// TIA Portal project "V6_V2.0" (V16)

(* hardware
DEVICE "S7-1200 station_1"  S7-1200 Station
   slot 0: "Rack_0"  S7-1200 Rack  Rack  V1.0
   slot 1: "PLC_Slave"  CPU 1214C DC/DC/DC  6ES7 214-1AG40-0XB0  V4.4
   slot 2: "DI 8/DQ 8x24VDC_1"  6ES7 223-1BH32-0XB0  V2.0
   slot 101: "CM 1241 (RS422/485)_1"  6ES7 241-1CH32-0XB0  V2.2
   slot 102: "CM 1241 (RS422/485)_2"  6ES7 241-1CH32-0XB0  V2.2
   slot 103: "CM 1241 (RS422/485)_3"  6ES7 241-1CH32-0XB0  V2.2
DEVICE "ADMIN_CONTROL_SYSTEM"  KTP700 Basic PN
   slot 0: "HMI_1"  KTP700 Basic PN  6AV2 123-2GB03-0AX0  15.1.0.0
   slot 1: "HMI_RT_1"  KTP700 Basic PN  6AV2 123-2GB03-0AX0  15.1.0.0
   slot 5: "HMI_1.IE_CP_1"  PROFINET Interface  15.0.1.0
      slot 1: "PROFINET Interface_1"  PROFINET Interface
         slot 1: "Port_1"  Port
DEVICE "PC_SEVER"  SIMATIC PC station
   slot 0: "SIMATIC PC station"  Rail  SIMATIC PC-Station  V1.0
      slot 125: "Stationmanager"  Station_Manager  V6.0.4
   slot 1: "HMI_RT_2"  WinCC RT Professional  6AV2 105-0xxxx-xxxx  16.0.0.0
   slot 2: "IE general_1"  IE General  IE_CP  V8.2.0
*)

// ===== PLC "PLC_Slave"  CPU 1214C DC/DC/DC =====

VAR_GLOBAL   // PLC tag table "Default tag table"
   "Sensor_Coun" AT %M100.0 : Bool;
   "Sensor_coun_Check" AT %M100.1 : Bool;
   "Tag_1" AT %I20.1 : Bool;
END_VAR

VAR_GLOBAL   // PLC tag table "SS"
   "SS01" AT %I0.1 : Bool;   // ht tren
   "SS02" AT %I0.2 : Bool;
   "SS03" AT %I0.3 : Bool;   // thang_ngan
   "SS04" AT %I0.4 : Bool;   // thang_dai
   "SS05" AT %I0.5 : Bool;
   "SS06" AT %I0.6 : Bool;
   "SS07" AT %I0.7 : Bool;   // mam_Chot_duoi
   "SS08" AT %I1.0 : Bool;   // mam_chot_tren
   "SS09" AT %I1.1 : Bool;
   "SS10" AT %I1.2 : Bool;
   "SS11" AT %I1.3 : Bool;
   "SS12" AT %I1.4 : Bool;   // xoay_trong
   "SS13" AT %I1.5 : Bool;   // xoay_ngoai
   "SS14" AT %I1.6 : Bool;
   "SS15" AT %I1.7 : Bool;
   "NANG" AT %Q0.1 : Bool;
   "XOAY" AT %Q0.0 : Bool;
   "SS00" AT %I0.0 : Bool;   // ht duoi
   "SS16" AT %I2.0 : Bool;
   "SS17" AT %I2.1 : Bool;
   "SS18" AT %I2.2 : Bool;
   "SS19" AT %I2.3 : Bool;
   "SS20" AT %I2.4 : Bool;
END_VAR

DATA_BLOCK "ControlSystems_DB"   // DB10
{ S7_Optimized_Access := 'FALSE' }
VERSION : 0.1
// stored: InstanceOfName ControlSystems
"ControlSystems"
BEGIN
END_DATA_BLOCK

DATA_BLOCK "MANUAL_DB"   // DB11
{ S7_Optimized_Access := 'TRUE' }
VERSION : 0.1
// stored: InstanceOfName MANUAL
"MANUAL"
BEGIN
END_DATA_BLOCK

DATA_BLOCK "AUTO_DB"   // DB12
{ S7_Optimized_Access := 'TRUE' }
VERSION : 0.1
// stored: InstanceOfName AUTO
"AUTO"
BEGIN
END_DATA_BLOCK

DATA_BLOCK "AutoMode1_DB"   // DB20
{ S7_Optimized_Access := 'TRUE' }
VERSION : 0.1
// stored: InstanceOfName AutoMode1
"AutoMode1"
BEGIN
END_DATA_BLOCK

DATA_BLOCK "AutoMode2_DB"   // DB21
{ S7_Optimized_Access := 'TRUE' }
VERSION : 0.1
// stored: InstanceOfName AutoMode2
"AutoMode2"
BEGIN
END_DATA_BLOCK

DATA_BLOCK "DataSetUp"   // DB24
{ S7_Optimized_Access := 'FALSE' }
VERSION : 0.1
   VAR
      SPEED : Struct
         ELEVATOR : Struct
            Speed_RunManual : Int := 500;
            Speed_StartUp : Int := 500;
            Speed_R1 : Int;
            Speed_R2 : Int;
            Speed_Stop : Int;
         END_STRUCT;
         Cart_Pallet : Struct
            Speed_RunManual : Int := 500;
            Speed_StartUp : Int := 500;
            Speed_R1 : Int;
            Speed_R2 : Int;
            Speed_Stop : Int;
         END_STRUCT;
      END_STRUCT;
      MODE : Struct
         Manual_Auto : Bool;
         ModeNumber : Int;
         AUTO : Struct
            "Auto/Mode1_Mode2" : Bool;
            MODE2 : Struct
               "Mode2/Mode1_Mode2" : Bool;
            END_STRUCT;
         END_STRUCT;
      END_STRUCT;
      DATA__STATUS_MODBUSRTU : Struct
         ELAVATOR : Struct
            StatusUp : Word := 16#0004;
            StartusDown : Word := 16#0002;
         END_STRUCT;
         CART : Struct
            StatusUp : Word := 16#0004;
            StartusDown : Word := 16#0002;
         END_STRUCT;
      END_STRUCT;
   END_VAR
BEGIN
END_DATA_BLOCK

DATA_BLOCK "ControlAtElevator_DB"   // DB25
{ S7_Optimized_Access := 'FALSE' }
VERSION : 0.1
// stored: InstanceOfName ControlAtElevator
"ControlAtElevator"
BEGIN
END_DATA_BLOCK

DATA_BLOCK "Data_ADMIN_HMI"   // DB26
{ S7_Optimized_Access := 'FALSE' }
VERSION : 0.1
   VAR
      OKE : Bool;
      blink_Manual : Bool;
      blink_Auto : Bool;
      blink_Cancel : Bool;
      blink_Setup : Bool;
      blink_Back : Bool;
      blink_Position : Bool;
      Position : Struct
         "201" : Bool;
         "202" : Bool;
         "101" : Bool;
         "102" : Bool;
      END_STRUCT;
      CheckPosition : Struct
         "201" : Bool;
         "202" : Bool;
         "101" : Bool;
         "102" : Bool;
      END_STRUCT;
      PositionNumber : Int;
   END_VAR
BEGIN
END_DATA_BLOCK

DATA_BLOCK "POSITION_DB"   // DB27
{ S7_Optimized_Access := 'TRUE' }
VERSION : 0.1
// stored: InstanceOfName POSITION
"POSITION"
BEGIN
END_DATA_BLOCK

DATA_BLOCK "ModbusRtu_DB"   // DB63
{ S7_Optimized_Access := 'TRUE' }
VERSION : 0.1
// stored: InstanceOfName ModbusRtu
"ModbusRtu"
BEGIN
END_DATA_BLOCK

DATA_BLOCK "FunctionsControlSystems_DB"   // DB65
{ S7_Optimized_Access := 'TRUE' }
VERSION : 0.1
// stored: InstanceOfName FunctionsControlSystems
"FunctionsControlSystems"
BEGIN
END_DATA_BLOCK

// folder: Control

DATA_BLOCK "Data_Control"   // DB5
{ S7_Optimized_Access := 'FALSE' }
VERSION : 0.1
   VAR
      AUTO : Struct
         "Auto.Mode1" : Struct
            STEP_E : Int;
            STEP_HP : Int;
            STEP_TR : Int;
         END_STRUCT;
         "Auto.Mode2_Mode1" : Struct
            Step_ParkingCar : Int;
            Step_GetCar : Int;
         END_STRUCT;
      END_STRUCT;
      Stop : Bool;
      START : Bool;
      RST : Bool;
      Auto_Manual : Bool;
      "Auto.Mode1_Mode2" : Bool;
      "Auto.Mode2_Mode1" : Bool;
      ERROR : Bool;
      ERRORNumber : Int;
      ModeAction : Int;
      ModeNumber : Int;
      SlotIDFrom : Int;
      SlotIDTO : Int;
      Lock : Bool;
      "Auto.ACTION" : Struct
         Elevator : Bool;
         Elevator_2 : Bool;
         HookPallet : Bool;
         HookPallet_2 : Bool;
         TableRotation : Bool;
         TableRotation_2 : Bool;
      END_STRUCT;
      Elevator : Struct
         Start : Bool;
         Done : Bool;
         Running : Bool;
         Error : Bool;
         UP : Bool;
         DOWN : Bool;
         SpeedManual : Int := 500;
         SpeedStartup : Int := 700;   // 7
         Speed1_Auto : Int := 2500;   // 25
         Speed2_Auto : Int := 1000;   // 10
         SpeedStop : Int := 500;   // 5
         "Step" : Int;
         DataSPEEDLift_INVT : Int;
         DataSTATUSControl_INVT : Word;
         DataStatusUPControl_Setup : Word := 16#0004;
         DataStatusDOWNControl_Setup : Word := 16#0002;
         FloorAddressControlNumber : Int := 1;
         FloorAddressControlNumber_Check : Int;
         FloorAddressReal : Int := 1;
         FloorAddressReal_Check : Int := 1;
         FloorAddressReal_Sub_FloorAddressControlNumber : Int;
         time_Run_one : Time := T#2s;   // 2s
         time_Run_Two : Time := T#8s;   // 8s
         time_Run_Three : Time;
      END_STRUCT;
      HookPallet : Struct
         Start : Bool;
         Done : Bool;
         Running : Bool;
         "1" : Bool;
         "2" : Bool;
         PositionControlNumber : Int;
         SpeedManual : Int := 500;
         SpeedStartup : Int := 2000;
         Speed1_Auto : Int := 3000;
         Speed2_Auto : Int := 2500;
         Speed3_Auto : Int := 1500;
         Speed4_Auto : Int := 500;
         time_Run_one : Time := T#7s;
         time_Run_Two : Time := T#11s;
         time_Run_Three : Time := T#5s;
         time_Run_Four : Time := T#2s;
         time_Run_Five : Time := T#2s;
         "Step" : Int;
         DataStatus1Control_Setup : Word := 16#0002;
         DataStatus2Control_Setup : Word := 16#0004;
         DataSPEEDLift_INVT : Int;
         DataSTATUSControl_INVT : Word;
         Current : Int;
         Volt : Int;
         Hz : Int;
      END_STRUCT;
      TableRotation : Struct
         UP : Struct
            Start : Bool;
            Running : Bool;
            Done : Bool;
            "Step" : Int;
            SpeedManual : Int := 1000;
            SpeedStart : Int := 5000;
            SpeedStop : Int := 1000;
            time1 : Time := T#5S_500MS;
         END_STRUCT;
         Down : Struct
            "Step" : Int;
            Running : Bool;
            Done : Bool;
            Start : Bool;
            SpeedManual : Int := 1000;
            SpeedStart : Int := 5000;
            SpeedStop : Int := 1000;
            time1 : Time := T#5S_500MS;
         END_STRUCT;
         Ro : Struct
            "Step" : Int;
            Running : Bool;
            Done : Bool;
            Start : Bool;
            SpeedManual : Int := 1000;
            SpeedStart : Int := 1000;
            Speed1 : Int := 5000;
            Speed2 : Int := 3500;
            Speed3 : Int := 1000;
            SpeedStop : Int := 300;
            time1 : Time := T#1s;
            time2 : Time := T#11s;
            time3 : Time := T#3s;
         END_STRUCT;
         DataSTATUSDown : Word := 16#0002;
         DataSTATUSUp : Word := 16#0004;
         Up_Manual : Bool;
         Down_Manual : Bool;
         "Ro.1_Manual" : Bool;
         "Ro.2_Manual" : Bool;
         DataSpeedINVT : Int;
         DataSpeedINVT_Ro : Int;
         DataSpeedINVT_Down_Up : Int;
         DataStatusINVT : Word;
         Running : Bool;
         Done : Bool;
         Current_Ro : Int;
         Current_Up_Down : Int;
         Current : Int;
         Volt_Ro : Int;
         Volt : Int;
         Volt_Up_Down : Int;
         HZ_Ro : Int;
         HZ : Int;
         HZ_Up_Down : Int;
      END_STRUCT;
      POSITION : Struct
         "201" : Bool;
         "202" : Bool;
         "201_C" : Bool;
         "202_C" : Bool;
         POSITIONumber : Int;
         Parking_Get : Bool;
      END_STRUCT;
   END_VAR
BEGIN
END_DATA_BLOCK

DATA_BLOCK "Data_mb_E"   // DB29
{ S7_Optimized_Access := 'FALSE' }
VERSION : 0.1
   VAR
      Data_Mb : Struct
         Hz : Int;
         Current : Int;
         Volt : Int;
      END_STRUCT;
   END_VAR
BEGIN
END_DATA_BLOCK

DATA_BLOCK "Data_mb_T"   // DB30
{ S7_Optimized_Access := 'FALSE' }
VERSION : 0.1
   VAR
      Data_Mb : Struct
         Hz : Int;
         Current : Int;
         Volt : Int;
      END_STRUCT;
   END_VAR
BEGIN
END_DATA_BLOCK

DATA_BLOCK "Data_MB_R"   // DB31
{ S7_Optimized_Access := 'FALSE' }
VERSION : 0.1
   VAR
      Data_Mb : Struct
         Hz : Int;
         Current : Int;
         Volt : Int;
      END_STRUCT;
   END_VAR
BEGIN
END_DATA_BLOCK

// folder: Control/FunctionsControlSystem

DATA_BLOCK "HookPalletMcFullFunction_DB"   // DB6
{ S7_Optimized_Access := 'TRUE' }
VERSION : 0.1
// stored: InstanceOfName HookPalletMcFullFunction
"HookPalletMcFullFunction"
BEGIN
END_DATA_BLOCK

DATA_BLOCK "TableRotationPalletMCFullFunction_DB"   // DB7
{ S7_Optimized_Access := 'TRUE' }
VERSION : 0.1
// stored: InstanceOfName TableRotationPalletMCFullFunction
"TableRotationPalletMCFullFunction"
BEGIN
END_DATA_BLOCK

DATA_BLOCK "TableRotationPalletMCFullFunction_DB_1"   // DB9
{ S7_Optimized_Access := 'TRUE' }
VERSION : 0.1
// stored: InstanceOfName TableRotationPalletMCFullFunction
"TableRotationPalletMCFullFunction"
BEGIN
END_DATA_BLOCK

DATA_BLOCK "TableRotationPalletMCFullFunction_DB_2"   // DB28
{ S7_Optimized_Access := 'TRUE' }
VERSION : 0.1
// stored: InstanceOfName TableRotationPalletMCFullFunction
"TableRotationPalletMCFullFunction"
BEGIN
END_DATA_BLOCK

DATA_BLOCK "LIFT_Full_Function_DB_1"   // DB66
{ S7_Optimized_Access := 'FALSE' }
VERSION : 0.1
// stored: InstanceOfName ElevatorMcFullFunction
"ElevatorMcFullFunction"
BEGIN
END_DATA_BLOCK

// folder: Control/Modbus RTU/Modbus RTU_Lift

DATA_BLOCK "Modbus_RTU_V1.0_DB_Lift"   // DB1
{ S7_Optimized_Access := 'FALSE' }
VERSION : 0.1
// stored: InstanceOfName Modbus_RTU_V1.0_Lift
"Modbus_RTU_V1.0_Lift"
BEGIN
END_DATA_BLOCK

DATA_BLOCK "Data_Modbus_RTU_Lift"   // DB4
{ S7_Optimized_Access := 'FALSE' }
VERSION : 0.1
   VAR
      "Modbus_Comm_Load-" : Struct
         Done : Bool;
         Req : Bool;
         Error : Bool;
         Busy : Bool;
         Status : Word;
      END_STRUCT;
      Modbus_Master : Struct
         Done : Bool;
         Req : Bool;
         mode : Int := 0;
         mode1 : Int := 1;
         Error : Bool;
         Busy : Bool;
         Status : Word;
      END_STRUCT;
      Address_INVT : Int := 4;
      "Step" : Int;
      Address_Status : UInt := 40009;
      Address_Speed : UInt := 40014;
      Address_Current_HZ_Volt : UInt := 40201;
      Error_Check_Number : Int;
      RST_error_Modbus : Bool;
   END_VAR
BEGIN
END_DATA_BLOCK

// folder: Control/Modbus RTU/Modbus_RTU_Ro

DATA_BLOCK "Data_Modbus_RTU_Ro"   // DB8
{ S7_Optimized_Access := 'FALSE' }
VERSION : 0.1
   VAR
      "Modbus_Comm_Load-" : Struct
         Done : Bool;
         Req : Bool;
         Error : Bool;
         Busy : Bool;
         Status : Word;
      END_STRUCT;
      Modbus_Master : Struct
         Done : Bool;
         Req : Bool;
         Error : Bool;
         Busy : Bool;
         Status : Word;
      END_STRUCT;
      Address_INVT : Int := 2;
      "Step" : Int;
      Address_Status : UInt := 40009;
      Address_Speed : UInt := 40014;
      Address_Current_HZ_Volt : UInt := 40201;
      Address_Volt : UInt;
      Address_Hz : UInt;
      Error_Check_Number : Int;
      RST_error_Modbus : Bool;
   END_VAR
BEGIN
END_DATA_BLOCK

DATA_BLOCK "Modbus_RTU_V1.0_Ro_DB"   // DB13
{ S7_Optimized_Access := 'FALSE' }
VERSION : 0.1
// stored: InstanceOfName Modbus_RTU_V1.0_Ro
"Modbus_RTU_V1.0_Ro"
BEGIN
END_DATA_BLOCK

// folder: Control/Modbus RTU/Modbus_RTU_Tray

DATA_BLOCK "Data_Modbus_RTU_Tray"   // DB14
{ S7_Optimized_Access := 'FALSE' }
VERSION : 0.1
   VAR
      "Modbus_Comm_Load-" : Struct
         Done : Bool;
         Req : Bool;
         Error : Bool;
         Busy : Bool;
         Status : Word;
      END_STRUCT;
      Modbus_Master : Struct
         Done : Bool;
         Req : Bool;
         Error : Bool;
         Busy : Bool;
         Status : Word;
      END_STRUCT;
      Address_INVT : Int := 3;
      "Step" : Int;
      Address_Status : UInt := 40009;
      ADDR_Resistor_Current_HZ_Volt : UInt := 40201;
      Address_Speed : UInt := 40014;
      Error_Check_Number : Int;
      RST_error_Modbus : Bool;
   END_VAR
BEGIN
END_DATA_BLOCK

DATA_BLOCK "Modbus_RTU_V1.0_Tray_DB"   // DB15
{ S7_Optimized_Access := 'FALSE' }
VERSION : 0.1
// stored: InstanceOfName Modbus_RTU_V1.0_Tray
"Modbus_RTU_V1.0_Tray"
BEGIN
END_DATA_BLOCK

// folder: System blocks/Program resources

DATA_BLOCK "IEC_Timer_0_DB"   // DB22
{ S7_Optimized_Access := 'TRUE' }
AUTHOR : Simatic
FAMILY : IEC
NAME : IEC_TMR
VERSION : 1.0
// stored: InstanceOfName IEC_TIMER
"IEC_TIMER"
BEGIN
END_DATA_BLOCK

DATA_BLOCK "IEC_Timer_0_DB_1"   // DB41
{ S7_Optimized_Access := 'TRUE' }
AUTHOR : Simatic
FAMILY : IEC
NAME : IEC_TMR
VERSION : 1.0
// stored: InstanceOfName IEC_TIMER
"IEC_TIMER"
BEGIN
END_DATA_BLOCK

DATA_BLOCK "IEC_Timer_0_DB_2"   // DB42
{ S7_Optimized_Access := 'TRUE' }
AUTHOR : Simatic
FAMILY : IEC
NAME : IEC_TMR
VERSION : 1.0
// stored: InstanceOfName IEC_TIMER
"IEC_TIMER"
BEGIN
END_DATA_BLOCK

DATA_BLOCK "IEC_Timer_0_DB_3"   // DB43
{ S7_Optimized_Access := 'TRUE' }
AUTHOR : Simatic
FAMILY : IEC
NAME : IEC_TMR
VERSION : 1.0
// stored: InstanceOfName IEC_TIMER
"IEC_TIMER"
BEGIN
END_DATA_BLOCK

DATA_BLOCK "IEC_Timer_0_DB_4"   // DB44
{ S7_Optimized_Access := 'TRUE' }
AUTHOR : Simatic
FAMILY : IEC
NAME : IEC_TMR
VERSION : 1.0
// stored: InstanceOfName IEC_TIMER
"IEC_TIMER"
BEGIN
END_DATA_BLOCK

DATA_BLOCK "IEC_Timer_0_DB_6"   // DB46
{ S7_Optimized_Access := 'TRUE' }
AUTHOR : Simatic
FAMILY : IEC
NAME : IEC_TMR
VERSION : 1.0
// stored: InstanceOfName IEC_TIMER
"IEC_TIMER"
BEGIN
END_DATA_BLOCK

DATA_BLOCK "IEC_Timer_0_DB_5"   // DB48
{ S7_Optimized_Access := 'TRUE' }
AUTHOR : Simatic
FAMILY : IEC
NAME : IEC_TMR
VERSION : 1.0
// stored: InstanceOfName IEC_TIMER
"IEC_TIMER"
BEGIN
END_DATA_BLOCK

DATA_BLOCK "IEC_Timer_0_DB_7"   // DB49
{ S7_Optimized_Access := 'TRUE' }
AUTHOR : Simatic
FAMILY : IEC
NAME : IEC_TMR
VERSION : 1.0
// stored: InstanceOfName IEC_TIMER
"IEC_TIMER"
BEGIN
END_DATA_BLOCK

DATA_BLOCK "IEC_Timer_0_DB_8"   // DB50
{ S7_Optimized_Access := 'TRUE' }
AUTHOR : Simatic
FAMILY : IEC
NAME : IEC_TMR
VERSION : 1.0
// stored: InstanceOfName IEC_TIMER
"IEC_TIMER"
BEGIN
END_DATA_BLOCK

DATA_BLOCK "IEC_Timer_0_DB_9"   // DB51
{ S7_Optimized_Access := 'TRUE' }
AUTHOR : Simatic
FAMILY : IEC
NAME : IEC_TMR
VERSION : 1.0
// stored: InstanceOfName IEC_TIMER
"IEC_TIMER"
BEGIN
END_DATA_BLOCK

DATA_BLOCK "IEC_Timer_0_DB_10"   // DB52
{ S7_Optimized_Access := 'TRUE' }
AUTHOR : Simatic
FAMILY : IEC
NAME : IEC_TMR
VERSION : 1.0
// stored: InstanceOfName IEC_TIMER
"IEC_TIMER"
BEGIN
END_DATA_BLOCK

DATA_BLOCK "IEC_Timer_0_DB_11"   // DB53
{ S7_Optimized_Access := 'TRUE' }
AUTHOR : Simatic
FAMILY : IEC
NAME : IEC_TMR
VERSION : 1.0
// stored: InstanceOfName IEC_TIMER
"IEC_TIMER"
BEGIN
END_DATA_BLOCK

DATA_BLOCK "IEC_Timer_0_DB_12"   // DB54
{ S7_Optimized_Access := 'TRUE' }
AUTHOR : Simatic
FAMILY : IEC
NAME : IEC_TMR
VERSION : 1.0
// stored: InstanceOfName IEC_TIMER
"IEC_TIMER"
BEGIN
END_DATA_BLOCK

DATA_BLOCK "IEC_Timer_0_DB_13"   // DB55
{ S7_Optimized_Access := 'TRUE' }
AUTHOR : Simatic
FAMILY : IEC
NAME : IEC_TMR
VERSION : 1.0
// stored: InstanceOfName IEC_TIMER
"IEC_TIMER"
BEGIN
END_DATA_BLOCK

DATA_BLOCK "IEC_Timer_0_DB_17"   // DB61
{ S7_Optimized_Access := 'TRUE' }
AUTHOR : Simatic
FAMILY : IEC
NAME : IEC_TMR
VERSION : 1.0
// stored: InstanceOfName IEC_TIMER
"IEC_TIMER"
BEGIN
END_DATA_BLOCK

DATA_BLOCK "IEC_Timer_0_DB_19"   // DB64
{ S7_Optimized_Access := 'TRUE' }
AUTHOR : Simatic
FAMILY : IEC
NAME : IEC_TMR
VERSION : 1.0
// stored: InstanceOfName IEC_TIMER
"IEC_TIMER"
BEGIN
END_DATA_BLOCK

DATA_BLOCK "IEC_Timer_0_DB_21"   // DB67
{ S7_Optimized_Access := 'TRUE' }
AUTHOR : Simatic
FAMILY : IEC
NAME : IEC_TMR
VERSION : 1.0
// stored: InstanceOfName IEC_TIMER
"IEC_TIMER"
BEGIN
END_DATA_BLOCK

// folder: (top level)

FUNCTION_BLOCK "ControlSystems"   // FB2, LAD
{ S7_Optimized_Access := 'FALSE' }
VERSION : 0.1
BEGIN

REGION Network 1
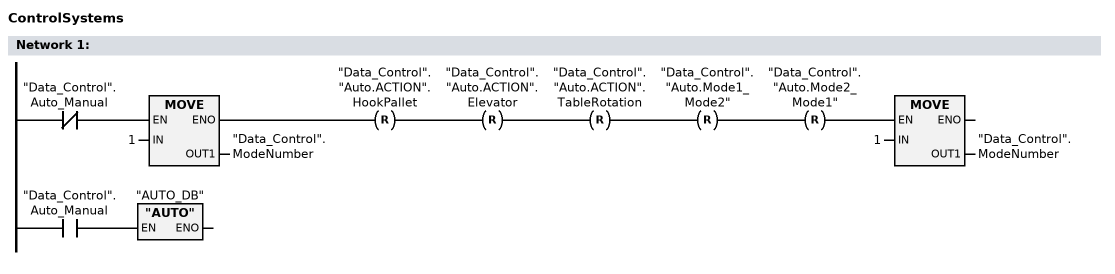
   RUNG wire#powerrail
      I_Contact( "Data_Control".Auto_Manual )
      Move(in := 1, out1 => "Data_Control".ModeNumber)
      R_Coil( "Data_Control"."Auto.ACTION".HookPallet )
      R_Coil( "Data_Control"."Auto.ACTION".Elevator )
      R_Coil( "Data_Control"."Auto.ACTION".TableRotation )
      R_Coil( "Data_Control"."Auto.Mode1_Mode2" )
      R_Coil( "Data_Control"."Auto.Mode2_Mode1" )
      Move(in := 1, out1 => "Data_Control".ModeNumber)
   END_RUNG
   RUNG wire#powerrail
      Contact( "Data_Control".Auto_Manual )
      "AUTO_DB"()
   END_RUNG
   // the same network as SCL:
   IF NOT "Data_Control".Auto_Manual THEN
       "Data_Control".ModeNumber := 1;
       "Data_Control"."Auto.ACTION".HookPallet := FALSE;
       "Data_Control"."Auto.ACTION".Elevator := FALSE;
       "Data_Control"."Auto.ACTION".TableRotation := FALSE;
       "Data_Control"."Auto.Mode1_Mode2" := FALSE;
       "Data_Control"."Auto.Mode2_Mode1" := FALSE;
       "Data_Control".ModeNumber := 1;
   END_IF;
   IF "Data_Control".Auto_Manual THEN
       "AUTO_DB"();   // "AUTO"
   END_IF;
END_REGION
END_FUNCTION_BLOCK

FUNCTION_BLOCK "MANUAL"   // FB3, LAD
{ S7_Optimized_Access := 'TRUE' }
VERSION : 0.1
BEGIN
END_FUNCTION_BLOCK

FUNCTION_BLOCK "AUTO"   // FB4, LAD
{ S7_Optimized_Access := 'TRUE' }
VERSION : 0.1
   VAR_TEMP   // added for the SCL form of the ladder/FBD networks
      _w1 : Bool;
      _w2 : Bool;
   END_VAR
BEGIN

REGION Network 1
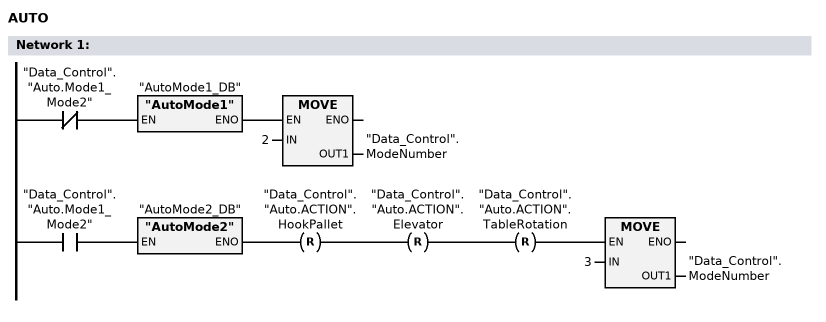
   RUNG wire#powerrail
      I_Contact( "Data_Control"."Auto.Mode1_Mode2" )
      "AutoMode1_DB"()
      Move(in := 2, out1 => "Data_Control".ModeNumber)
   END_RUNG
   RUNG wire#powerrail
      Contact( "Data_Control"."Auto.Mode1_Mode2" )
      "AutoMode2_DB"()
      R_Coil( "Data_Control"."Auto.ACTION".HookPallet )
      R_Coil( "Data_Control"."Auto.ACTION".Elevator )
      R_Coil( "Data_Control"."Auto.ACTION".TableRotation )
      Move(in := 3, out1 => "Data_Control".ModeNumber)
   END_RUNG
   // the same network as SCL:
   "AutoMode1_DB"(EN := NOT "Data_Control"."Auto.Mode1_Mode2", ENO => #_w1);   // "AutoMode1"
   IF #_w1 THEN "Data_Control".ModeNumber := 2; END_IF;
   "AutoMode2_DB"(EN := "Data_Control"."Auto.Mode1_Mode2", ENO => #_w2);   // "AutoMode2"
   IF #_w2 THEN
       "Data_Control"."Auto.ACTION".HookPallet := FALSE;
       "Data_Control"."Auto.ACTION".Elevator := FALSE;
       "Data_Control"."Auto.ACTION".TableRotation := FALSE;
       "Data_Control".ModeNumber := 3;
   END_IF;
END_REGION
END_FUNCTION_BLOCK

FUNCTION_BLOCK "AutoMode1"   // FB5, LAD
{ S7_Optimized_Access := 'TRUE' }
VERSION : 0.1
   VAR_TEMP   // added for the SCL form of the ladder/FBD networks
      _w1 : Bool;
   END_VAR
BEGIN

REGION Network 1
   // Elevator
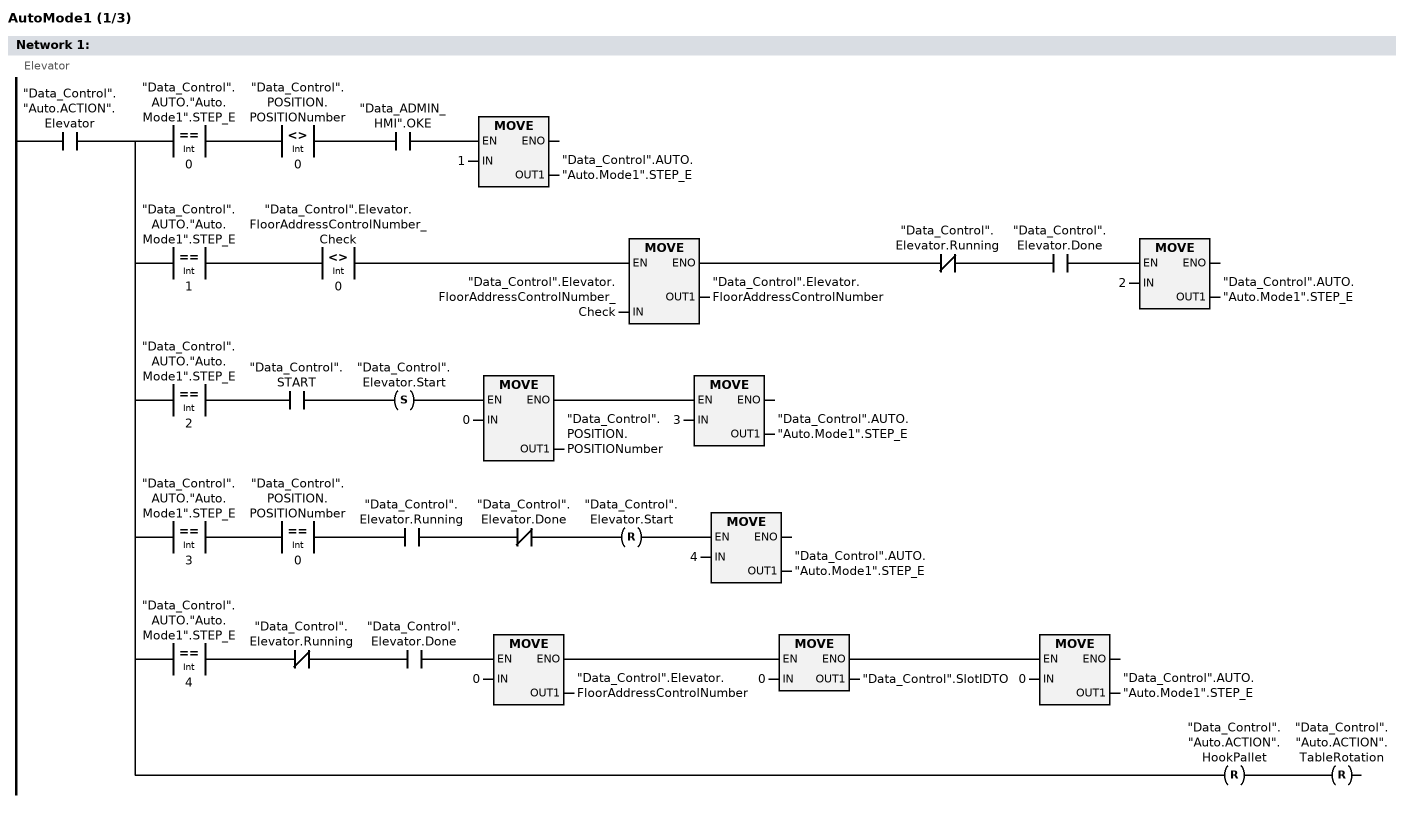
   RUNG wire#powerrail
      Contact( "Data_Control"."Auto.ACTION".Elevator )
      wire#w1
      { S7_Templates := "SrcType := Int" } EQ_Contact(in1 := "Data_Control".AUTO."Auto.Mode1".STEP_E, in2 := 0)
      { S7_Templates := "SrcType := Int" } NE_Contact(in1 := "Data_Control".POSITION.POSITIONumber, in2 := 0)
      Contact( "Data_ADMIN_HMI".OKE )
      Move(in := 1, out1 => "Data_Control".AUTO."Auto.Mode1".STEP_E)
   END_RUNG
   RUNG wire#w1
      { S7_Templates := "SrcType := Int" } EQ_Contact(in1 := "Data_Control".AUTO."Auto.Mode1".STEP_E, in2 := 1)
      { S7_Templates := "SrcType := Int" } NE_Contact(in1 := "Data_Control".Elevator.FloorAddressControlNumber_Check, in2 := 0)
      Move(in := "Data_Control".Elevator.FloorAddressControlNumber_Check, out1 => "Data_Control".Elevator.FloorAddressControlNumber)
      I_Contact( "Data_Control".Elevator.Running )
      Contact( "Data_Control".Elevator.Done )
      Move(in := 2, out1 => "Data_Control".AUTO."Auto.Mode1".STEP_E)
   END_RUNG
   RUNG wire#w1
      { S7_Templates := "SrcType := Int" } EQ_Contact(in1 := "Data_Control".AUTO."Auto.Mode1".STEP_E, in2 := 2)
      Contact( "Data_Control".START )
      S_Coil( "Data_Control".Elevator.Start )
      Move(in := 0, out1 => "Data_Control".POSITION.POSITIONumber)
      Move(in := 3, out1 => "Data_Control".AUTO."Auto.Mode1".STEP_E)
   END_RUNG
   RUNG wire#w1
      { S7_Templates := "SrcType := Int" } EQ_Contact(in1 := "Data_Control".AUTO."Auto.Mode1".STEP_E, in2 := 3)
      { S7_Templates := "SrcType := Int" } EQ_Contact(in1 := "Data_Control".POSITION.POSITIONumber, in2 := 0)
      Contact( "Data_Control".Elevator.Running )
      I_Contact( "Data_Control".Elevator.Done )
      R_Coil( "Data_Control".Elevator.Start )
      Move(in := 4, out1 => "Data_Control".AUTO."Auto.Mode1".STEP_E)
   END_RUNG
   RUNG wire#w1
      { S7_Templates := "SrcType := Int" } EQ_Contact(in1 := "Data_Control".AUTO."Auto.Mode1".STEP_E, in2 := 4)
      I_Contact( "Data_Control".Elevator.Running )
      Contact( "Data_Control".Elevator.Done )
      Move(in := 0, out1 => "Data_Control".Elevator.FloorAddressControlNumber)
      Move(in := 0, out1 => "Data_Control".SlotIDTO)
      Move(in := 0, out1 => "Data_Control".AUTO."Auto.Mode1".STEP_E)
   END_RUNG
   RUNG wire#w1
      R_Coil( "Data_Control"."Auto.ACTION".HookPallet )
      R_Coil( "Data_Control"."Auto.ACTION".TableRotation )
   END_RUNG
   // the same network as SCL:
   IF "Data_Control"."Auto.ACTION".Elevator AND ("Data_Control".AUTO."Auto.Mode1".STEP_E = 0) AND ("Data_Control".POSITION.POSITIONumber <> 0) AND "Data_ADMIN_HMI".OKE THEN
       "Data_Control".AUTO."Auto.Mode1".STEP_E := 1;
   END_IF;
   #_w1 := "Data_Control"."Auto.ACTION".Elevator AND ("Data_Control".AUTO."Auto.Mode1".STEP_E = 1) AND ("Data_Control".Elevator.FloorAddressControlNumber_Check <> 0);
   IF #_w1 THEN
       "Data_Control".Elevator.FloorAddressControlNumber := "Data_Control".Elevator.FloorAddressControlNumber_Check;
   END_IF;
   IF #_w1 AND NOT "Data_Control".Elevator.Running AND "Data_Control".Elevator.Done THEN
       "Data_Control".AUTO."Auto.Mode1".STEP_E := 2;
   END_IF;
   IF "Data_Control"."Auto.ACTION".Elevator AND ("Data_Control".AUTO."Auto.Mode1".STEP_E = 2) AND "Data_Control".START THEN
       "Data_Control".Elevator.Start := TRUE;
       "Data_Control".POSITION.POSITIONumber := 0;
       "Data_Control".AUTO."Auto.Mode1".STEP_E := 3;
   END_IF;
   IF "Data_Control"."Auto.ACTION".Elevator AND ("Data_Control".AUTO."Auto.Mode1".STEP_E = 3) AND ("Data_Control".POSITION.POSITIONumber = 0) AND "Data_Control".Elevator.Running AND NOT "Data_Control".Elevator.Done THEN
       "Data_Control".Elevator.Start := FALSE;
       "Data_Control".AUTO."Auto.Mode1".STEP_E := 4;
   END_IF;
   IF "Data_Control"."Auto.ACTION".Elevator AND ("Data_Control".AUTO."Auto.Mode1".STEP_E = 4) AND NOT "Data_Control".Elevator.Running AND "Data_Control".Elevator.Done THEN
       "Data_Control".Elevator.FloorAddressControlNumber := 0;
       "Data_Control".SlotIDTO := 0;
       "Data_Control".AUTO."Auto.Mode1".STEP_E := 0;
   END_IF;
   IF "Data_Control"."Auto.ACTION".Elevator THEN
       "Data_Control"."Auto.ACTION".HookPallet := FALSE;
       "Data_Control"."Auto.ACTION".TableRotation := FALSE;
   END_IF;
END_REGION

REGION Network 2
   // HookPallet
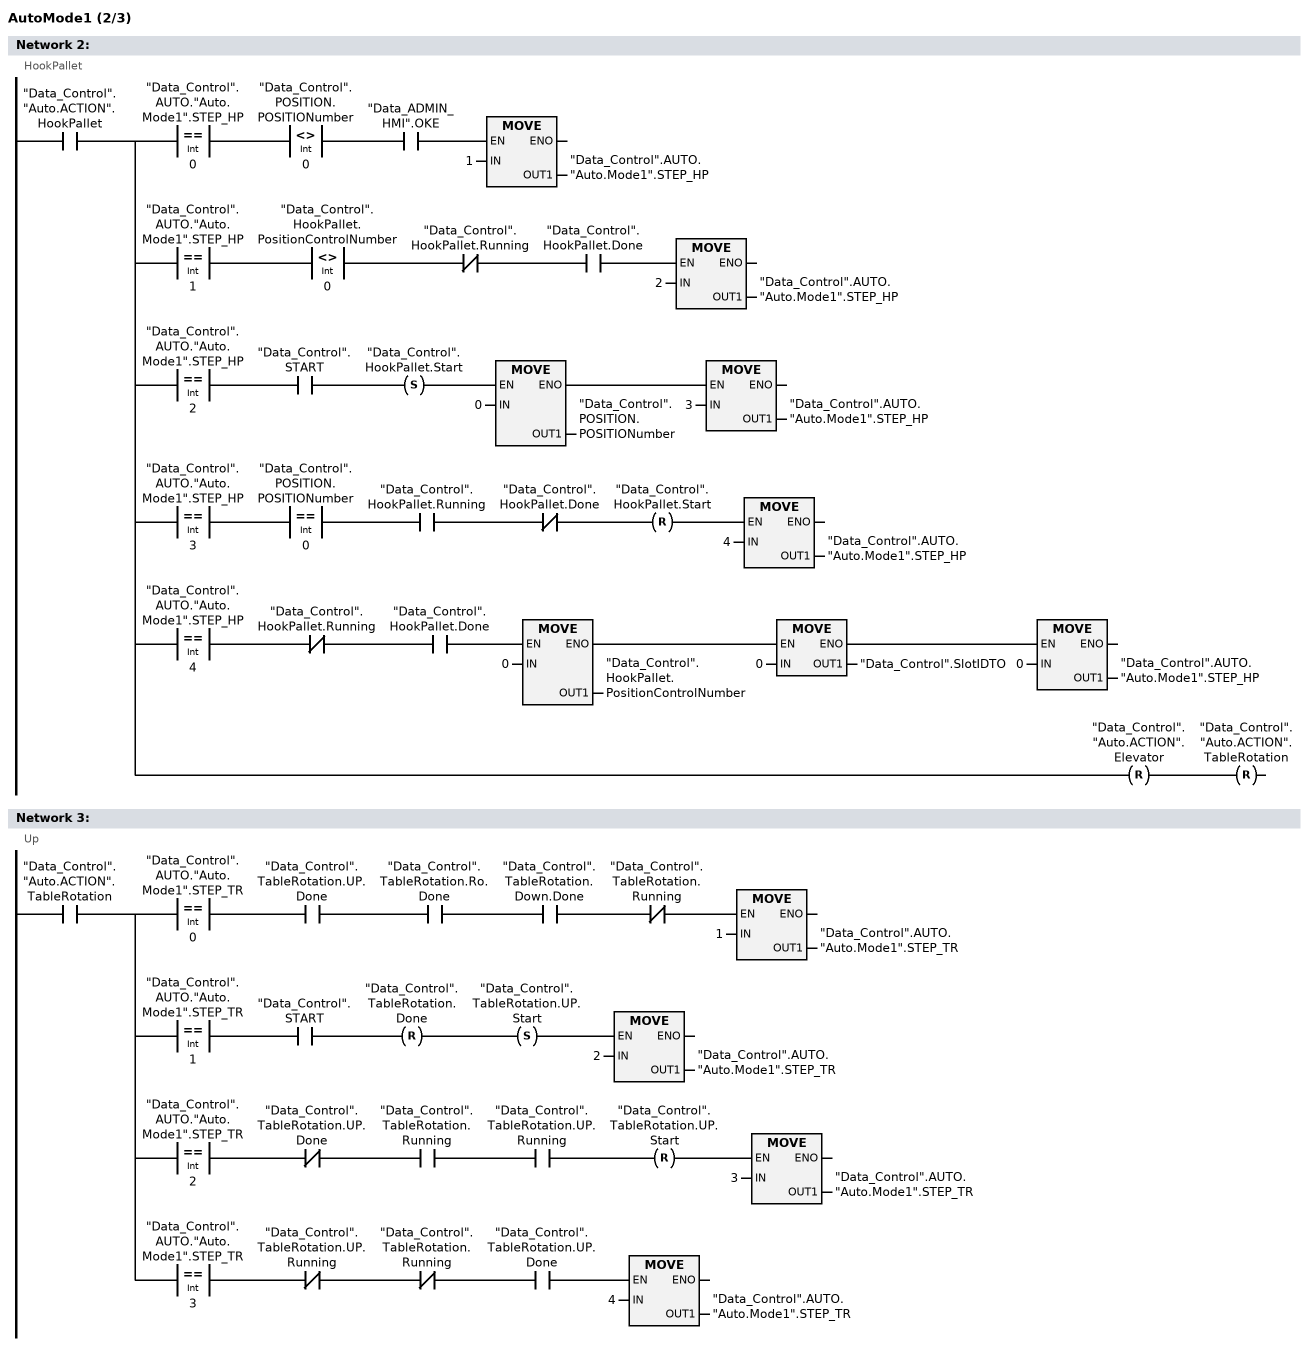
   RUNG wire#powerrail
      Contact( "Data_Control"."Auto.ACTION".HookPallet )
      wire#w1
      { S7_Templates := "SrcType := Int" } EQ_Contact(in1 := "Data_Control".AUTO."Auto.Mode1".STEP_HP, in2 := 0)
      { S7_Templates := "SrcType := Int" } NE_Contact(in1 := "Data_Control".POSITION.POSITIONumber, in2 := 0)
      Contact( "Data_ADMIN_HMI".OKE )
      Move(in := 1, out1 => "Data_Control".AUTO."Auto.Mode1".STEP_HP)
   END_RUNG
   RUNG wire#w1
      { S7_Templates := "SrcType := Int" } EQ_Contact(in1 := "Data_Control".AUTO."Auto.Mode1".STEP_HP, in2 := 1)
      { S7_Templates := "SrcType := Int" } NE_Contact(in1 := "Data_Control".HookPallet.PositionControlNumber, in2 := 0)
      I_Contact( "Data_Control".HookPallet.Running )
      Contact( "Data_Control".HookPallet.Done )
      Move(in := 2, out1 => "Data_Control".AUTO."Auto.Mode1".STEP_HP)
   END_RUNG
   RUNG wire#w1
      { S7_Templates := "SrcType := Int" } EQ_Contact(in1 := "Data_Control".AUTO."Auto.Mode1".STEP_HP, in2 := 2)
      Contact( "Data_Control".START )
      S_Coil( "Data_Control".HookPallet.Start )
      Move(in := 0, out1 => "Data_Control".POSITION.POSITIONumber)
      Move(in := 3, out1 => "Data_Control".AUTO."Auto.Mode1".STEP_HP)
   END_RUNG
   RUNG wire#w1
      { S7_Templates := "SrcType := Int" } EQ_Contact(in1 := "Data_Control".AUTO."Auto.Mode1".STEP_HP, in2 := 3)
      { S7_Templates := "SrcType := Int" } EQ_Contact(in1 := "Data_Control".POSITION.POSITIONumber, in2 := 0)
      Contact( "Data_Control".HookPallet.Running )
      I_Contact( "Data_Control".HookPallet.Done )
      R_Coil( "Data_Control".HookPallet.Start )
      Move(in := 4, out1 => "Data_Control".AUTO."Auto.Mode1".STEP_HP)
   END_RUNG
   RUNG wire#w1
      { S7_Templates := "SrcType := Int" } EQ_Contact(in1 := "Data_Control".AUTO."Auto.Mode1".STEP_HP, in2 := 4)
      I_Contact( "Data_Control".HookPallet.Running )
      Contact( "Data_Control".HookPallet.Done )
      Move(in := 0, out1 => "Data_Control".HookPallet.PositionControlNumber)
      Move(in := 0, out1 => "Data_Control".SlotIDTO)
      Move(in := 0, out1 => "Data_Control".AUTO."Auto.Mode1".STEP_HP)
   END_RUNG
   RUNG wire#w1
      R_Coil( "Data_Control"."Auto.ACTION".Elevator )
      R_Coil( "Data_Control"."Auto.ACTION".TableRotation )
   END_RUNG
   // the same network as SCL:
   IF "Data_Control"."Auto.ACTION".HookPallet AND ("Data_Control".AUTO."Auto.Mode1".STEP_HP = 0) AND ("Data_Control".POSITION.POSITIONumber <> 0) AND "Data_ADMIN_HMI".OKE THEN
       "Data_Control".AUTO."Auto.Mode1".STEP_HP := 1;
   END_IF;
   IF "Data_Control"."Auto.ACTION".HookPallet AND ("Data_Control".AUTO."Auto.Mode1".STEP_HP = 1) AND ("Data_Control".HookPallet.PositionControlNumber <> 0) AND NOT "Data_Control".HookPallet.Running AND "Data_Control".HookPallet.Done THEN
       "Data_Control".AUTO."Auto.Mode1".STEP_HP := 2;
   END_IF;
   IF "Data_Control"."Auto.ACTION".HookPallet AND ("Data_Control".AUTO."Auto.Mode1".STEP_HP = 2) AND "Data_Control".START THEN
       "Data_Control".HookPallet.Start := TRUE;
       "Data_Control".POSITION.POSITIONumber := 0;
       "Data_Control".AUTO."Auto.Mode1".STEP_HP := 3;
   END_IF;
   IF "Data_Control"."Auto.ACTION".HookPallet AND ("Data_Control".AUTO."Auto.Mode1".STEP_HP = 3) AND ("Data_Control".POSITION.POSITIONumber = 0) AND "Data_Control".HookPallet.Running AND NOT "Data_Control".HookPallet.Done THEN
       "Data_Control".HookPallet.Start := FALSE;
       "Data_Control".AUTO."Auto.Mode1".STEP_HP := 4;
   END_IF;
   IF "Data_Control"."Auto.ACTION".HookPallet AND ("Data_Control".AUTO."Auto.Mode1".STEP_HP = 4) AND NOT "Data_Control".HookPallet.Running AND "Data_Control".HookPallet.Done THEN
       "Data_Control".HookPallet.PositionControlNumber := 0;
       "Data_Control".SlotIDTO := 0;
       "Data_Control".AUTO."Auto.Mode1".STEP_HP := 0;
   END_IF;
   IF "Data_Control"."Auto.ACTION".HookPallet THEN
       "Data_Control"."Auto.ACTION".Elevator := FALSE;
       "Data_Control"."Auto.ACTION".TableRotation := FALSE;
   END_IF;
END_REGION

REGION Network 3
   // Up
   RUNG wire#powerrail
      Contact( "Data_Control"."Auto.ACTION".TableRotation )
      wire#w1
      { S7_Templates := "SrcType := Int" } EQ_Contact(in1 := "Data_Control".AUTO."Auto.Mode1".STEP_TR, in2 := 0)
      Contact( "Data_Control".TableRotation.UP.Done )
      Contact( "Data_Control".TableRotation.Ro.Done )
      Contact( "Data_Control".TableRotation.Down.Done )
      I_Contact( "Data_Control".TableRotation.Running )
      Move(in := 1, out1 => "Data_Control".AUTO."Auto.Mode1".STEP_TR)
   END_RUNG
   RUNG wire#w1
      { S7_Templates := "SrcType := Int" } EQ_Contact(in1 := "Data_Control".AUTO."Auto.Mode1".STEP_TR, in2 := 1)
      Contact( "Data_Control".START )
      R_Coil( "Data_Control".TableRotation.Done )
      S_Coil( "Data_Control".TableRotation.UP.Start )
      Move(in := 2, out1 => "Data_Control".AUTO."Auto.Mode1".STEP_TR)
   END_RUNG
   RUNG wire#w1
      { S7_Templates := "SrcType := Int" } EQ_Contact(in1 := "Data_Control".AUTO."Auto.Mode1".STEP_TR, in2 := 2)
      I_Contact( "Data_Control".TableRotation.UP.Done )
      Contact( "Data_Control".TableRotation.Running )
      Contact( "Data_Control".TableRotation.UP.Running )
      R_Coil( "Data_Control".TableRotation.UP.Start )
      Move(in := 3, out1 => "Data_Control".AUTO."Auto.Mode1".STEP_TR)
   END_RUNG
   RUNG wire#w1
      { S7_Templates := "SrcType := Int" } EQ_Contact(in1 := "Data_Control".AUTO."Auto.Mode1".STEP_TR, in2 := 3)
      I_Contact( "Data_Control".TableRotation.UP.Running )
      I_Contact( "Data_Control".TableRotation.Running )
      Contact( "Data_Control".TableRotation.UP.Done )
      Move(in := 4, out1 => "Data_Control".AUTO."Auto.Mode1".STEP_TR)
   END_RUNG
   // the same network as SCL:
   IF "Data_Control"."Auto.ACTION".TableRotation AND ("Data_Control".AUTO."Auto.Mode1".STEP_TR = 0) AND "Data_Control".TableRotation.UP.Done AND "Data_Control".TableRotation.Ro.Done AND "Data_Control".TableRotation.Down.Done AND NOT "Data_Control".TableRotation.Running THEN
       "Data_Control".AUTO."Auto.Mode1".STEP_TR := 1;
   END_IF;
   IF "Data_Control"."Auto.ACTION".TableRotation AND ("Data_Control".AUTO."Auto.Mode1".STEP_TR = 1) AND "Data_Control".START THEN
       "Data_Control".TableRotation.Done := FALSE;
       "Data_Control".TableRotation.UP.Start := TRUE;
       "Data_Control".AUTO."Auto.Mode1".STEP_TR := 2;
   END_IF;
   IF "Data_Control"."Auto.ACTION".TableRotation AND ("Data_Control".AUTO."Auto.Mode1".STEP_TR = 2) AND NOT "Data_Control".TableRotation.UP.Done AND "Data_Control".TableRotation.Running AND "Data_Control".TableRotation.UP.Running THEN
       "Data_Control".TableRotation.UP.Start := FALSE;
       "Data_Control".AUTO."Auto.Mode1".STEP_TR := 3;
   END_IF;
   IF "Data_Control"."Auto.ACTION".TableRotation AND ("Data_Control".AUTO."Auto.Mode1".STEP_TR = 3) AND NOT "Data_Control".TableRotation.UP.Running AND NOT "Data_Control".TableRotation.Running AND "Data_Control".TableRotation.UP.Done THEN
       "Data_Control".AUTO."Auto.Mode1".STEP_TR := 4;
   END_IF;
END_REGION

REGION Network 4
   // Ro
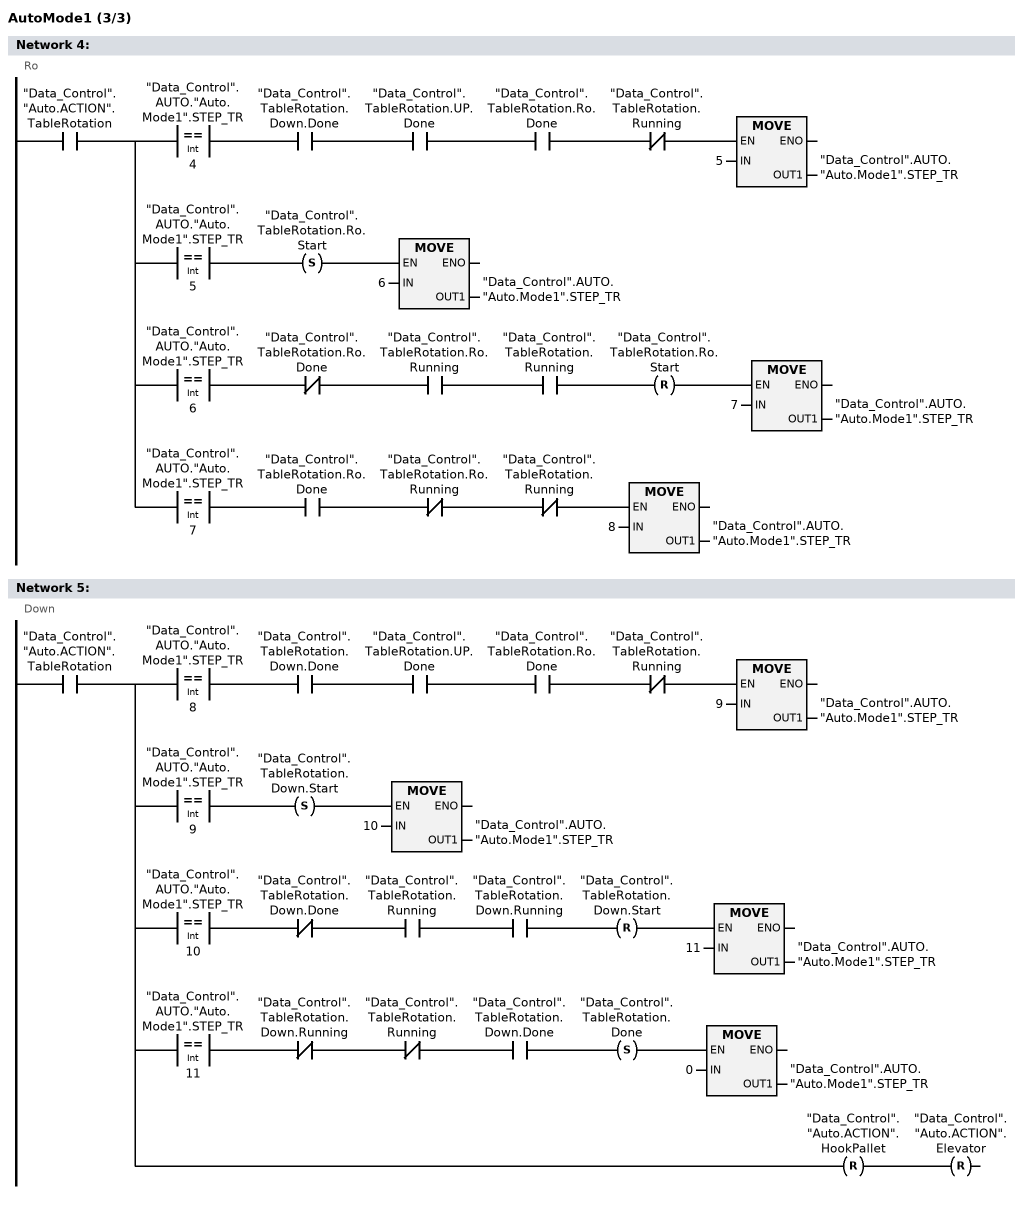
   RUNG wire#powerrail
      Contact( "Data_Control"."Auto.ACTION".TableRotation )
      wire#w1
      { S7_Templates := "SrcType := Int" } EQ_Contact(in1 := "Data_Control".AUTO."Auto.Mode1".STEP_TR, in2 := 4)
      Contact( "Data_Control".TableRotation.Down.Done )
      Contact( "Data_Control".TableRotation.UP.Done )
      Contact( "Data_Control".TableRotation.Ro.Done )
      I_Contact( "Data_Control".TableRotation.Running )
      Move(in := 5, out1 => "Data_Control".AUTO."Auto.Mode1".STEP_TR)
   END_RUNG
   RUNG wire#w1
      { S7_Templates := "SrcType := Int" } EQ_Contact(in1 := "Data_Control".AUTO."Auto.Mode1".STEP_TR, in2 := 5)
      S_Coil( "Data_Control".TableRotation.Ro.Start )
      Move(in := 6, out1 => "Data_Control".AUTO."Auto.Mode1".STEP_TR)
   END_RUNG
   RUNG wire#w1
      { S7_Templates := "SrcType := Int" } EQ_Contact(in1 := "Data_Control".AUTO."Auto.Mode1".STEP_TR, in2 := 6)
      I_Contact( "Data_Control".TableRotation.Ro.Done )
      Contact( "Data_Control".TableRotation.Ro.Running )
      Contact( "Data_Control".TableRotation.Running )
      R_Coil( "Data_Control".TableRotation.Ro.Start )
      Move(in := 7, out1 => "Data_Control".AUTO."Auto.Mode1".STEP_TR)
   END_RUNG
   RUNG wire#w1
      { S7_Templates := "SrcType := Int" } EQ_Contact(in1 := "Data_Control".AUTO."Auto.Mode1".STEP_TR, in2 := 7)
      Contact( "Data_Control".TableRotation.Ro.Done )
      I_Contact( "Data_Control".TableRotation.Ro.Running )
      I_Contact( "Data_Control".TableRotation.Running )
      Move(in := 8, out1 => "Data_Control".AUTO."Auto.Mode1".STEP_TR)
   END_RUNG
   // the same network as SCL:
   IF "Data_Control"."Auto.ACTION".TableRotation AND ("Data_Control".AUTO."Auto.Mode1".STEP_TR = 4) AND "Data_Control".TableRotation.Down.Done AND "Data_Control".TableRotation.UP.Done AND "Data_Control".TableRotation.Ro.Done AND NOT "Data_Control".TableRotation.Running THEN
       "Data_Control".AUTO."Auto.Mode1".STEP_TR := 5;
   END_IF;
   IF "Data_Control"."Auto.ACTION".TableRotation AND ("Data_Control".AUTO."Auto.Mode1".STEP_TR = 5) THEN
       "Data_Control".TableRotation.Ro.Start := TRUE;
       "Data_Control".AUTO."Auto.Mode1".STEP_TR := 6;
   END_IF;
   IF "Data_Control"."Auto.ACTION".TableRotation AND ("Data_Control".AUTO."Auto.Mode1".STEP_TR = 6) AND NOT "Data_Control".TableRotation.Ro.Done AND "Data_Control".TableRotation.Ro.Running AND "Data_Control".TableRotation.Running THEN
       "Data_Control".TableRotation.Ro.Start := FALSE;
       "Data_Control".AUTO."Auto.Mode1".STEP_TR := 7;
   END_IF;
   IF "Data_Control"."Auto.ACTION".TableRotation AND ("Data_Control".AUTO."Auto.Mode1".STEP_TR = 7) AND "Data_Control".TableRotation.Ro.Done AND NOT "Data_Control".TableRotation.Ro.Running AND NOT "Data_Control".TableRotation.Running THEN
       "Data_Control".AUTO."Auto.Mode1".STEP_TR := 8;
   END_IF;
END_REGION

REGION Network 5
   // Down
   RUNG wire#powerrail
      Contact( "Data_Control"."Auto.ACTION".TableRotation )
      wire#w1
      { S7_Templates := "SrcType := Int" } EQ_Contact(in1 := "Data_Control".AUTO."Auto.Mode1".STEP_TR, in2 := 8)
      Contact( "Data_Control".TableRotation.Down.Done )
      Contact( "Data_Control".TableRotation.UP.Done )
      Contact( "Data_Control".TableRotation.Ro.Done )
      I_Contact( "Data_Control".TableRotation.Running )
      Move(in := 9, out1 => "Data_Control".AUTO."Auto.Mode1".STEP_TR)
   END_RUNG
   RUNG wire#w1
      { S7_Templates := "SrcType := Int" } EQ_Contact(in1 := "Data_Control".AUTO."Auto.Mode1".STEP_TR, in2 := 9)
      S_Coil( "Data_Control".TableRotation.Down.Start )
      Move(in := 10, out1 => "Data_Control".AUTO."Auto.Mode1".STEP_TR)
   END_RUNG
   RUNG wire#w1
      { S7_Templates := "SrcType := Int" } EQ_Contact(in1 := "Data_Control".AUTO."Auto.Mode1".STEP_TR, in2 := 10)
      I_Contact( "Data_Control".TableRotation.Down.Done )
      Contact( "Data_Control".TableRotation.Running )
      Contact( "Data_Control".TableRotation.Down.Running )
      R_Coil( "Data_Control".TableRotation.Down.Start )
      Move(in := 11, out1 => "Data_Control".AUTO."Auto.Mode1".STEP_TR)
   END_RUNG
   RUNG wire#w1
      { S7_Templates := "SrcType := Int" } EQ_Contact(in1 := "Data_Control".AUTO."Auto.Mode1".STEP_TR, in2 := 11)
      I_Contact( "Data_Control".TableRotation.Down.Running )
      I_Contact( "Data_Control".TableRotation.Running )
      Contact( "Data_Control".TableRotation.Down.Done )
      S_Coil( "Data_Control".TableRotation.Done )
      Move(in := 0, out1 => "Data_Control".AUTO."Auto.Mode1".STEP_TR)
   END_RUNG
   RUNG wire#w1
      R_Coil( "Data_Control"."Auto.ACTION".HookPallet )
      R_Coil( "Data_Control"."Auto.ACTION".Elevator )
   END_RUNG
   // the same network as SCL:
   IF "Data_Control"."Auto.ACTION".TableRotation AND ("Data_Control".AUTO."Auto.Mode1".STEP_TR = 8) AND "Data_Control".TableRotation.Down.Done AND "Data_Control".TableRotation.UP.Done AND "Data_Control".TableRotation.Ro.Done AND NOT "Data_Control".TableRotation.Running THEN
       "Data_Control".AUTO."Auto.Mode1".STEP_TR := 9;
   END_IF;
   IF "Data_Control"."Auto.ACTION".TableRotation AND ("Data_Control".AUTO."Auto.Mode1".STEP_TR = 9) THEN
       "Data_Control".TableRotation.Down.Start := TRUE;
       "Data_Control".AUTO."Auto.Mode1".STEP_TR := 10;
   END_IF;
   IF "Data_Control"."Auto.ACTION".TableRotation AND ("Data_Control".AUTO."Auto.Mode1".STEP_TR = 10) AND NOT "Data_Control".TableRotation.Down.Done AND "Data_Control".TableRotation.Running AND "Data_Control".TableRotation.Down.Running THEN
       "Data_Control".TableRotation.Down.Start := FALSE;
       "Data_Control".AUTO."Auto.Mode1".STEP_TR := 11;
   END_IF;
   IF "Data_Control"."Auto.ACTION".TableRotation AND ("Data_Control".AUTO."Auto.Mode1".STEP_TR = 11) AND NOT "Data_Control".TableRotation.Down.Running AND NOT "Data_Control".TableRotation.Running AND "Data_Control".TableRotation.Down.Done THEN
       "Data_Control".TableRotation.Done := TRUE;
       "Data_Control".AUTO."Auto.Mode1".STEP_TR := 0;
   END_IF;
   IF "Data_Control"."Auto.ACTION".TableRotation THEN
       "Data_Control"."Auto.ACTION".HookPallet := FALSE;
       "Data_Control"."Auto.ACTION".Elevator := FALSE;
   END_IF;
END_REGION
END_FUNCTION_BLOCK

FUNCTION_BLOCK "AutoMode2"   // FB6, LAD
{ S7_Optimized_Access := 'TRUE' }
VERSION : 0.1
   VAR_TEMP   // added for the SCL form of the ladder/FBD networks
      _w1 : Bool;
      _w2 : Bool;
      _w3 : Bool;
      _w4 : Bool;
   END_VAR
BEGIN

REGION Network 1
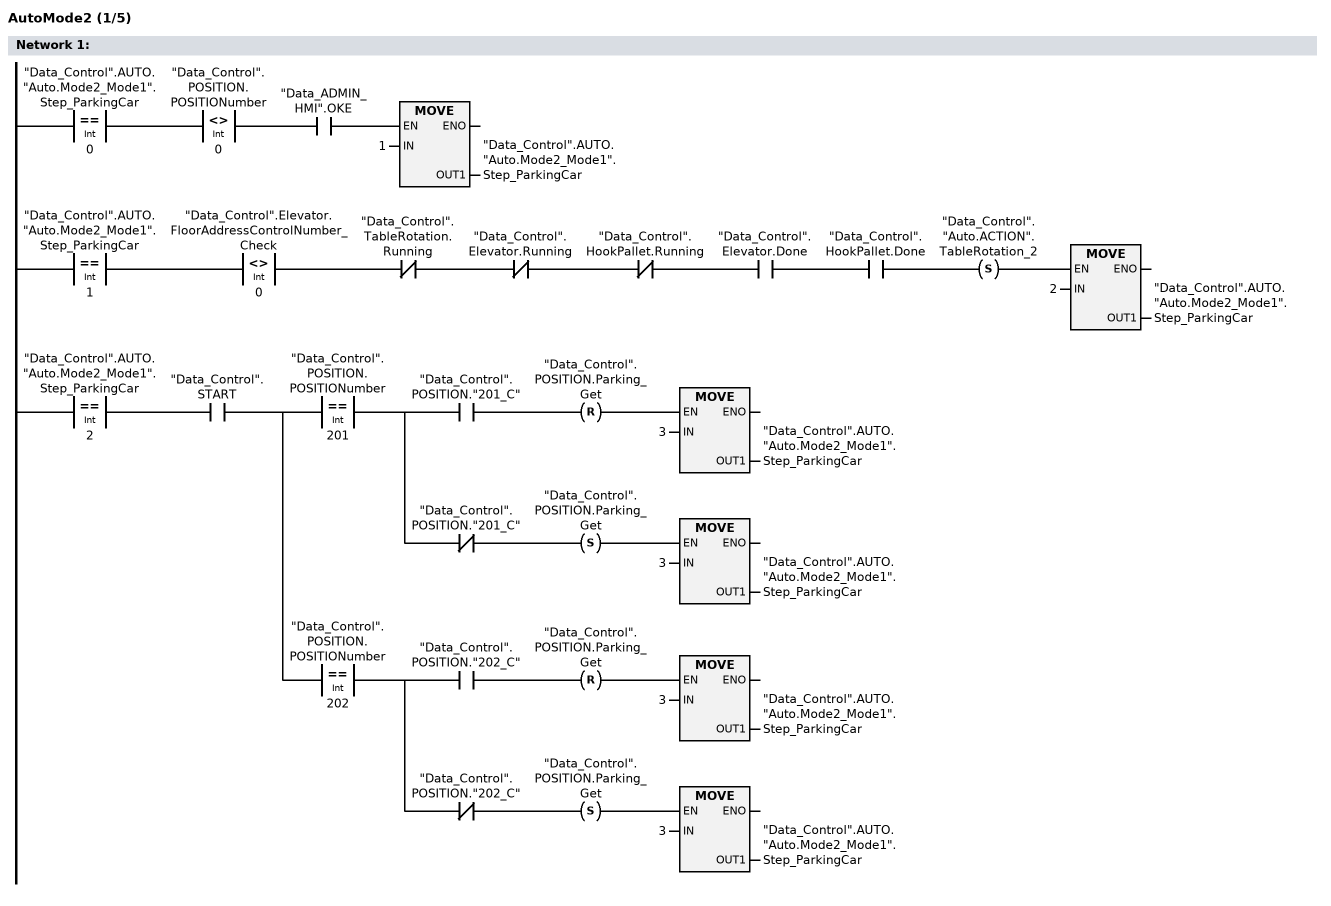
   RUNG wire#powerrail
      { S7_Templates := "SrcType := Int" } EQ_Contact(in1 := "Data_Control".AUTO."Auto.Mode2_Mode1".Step_ParkingCar, in2 := 0)
      { S7_Templates := "SrcType := Int" } NE_Contact(in1 := "Data_Control".POSITION.POSITIONumber, in2 := 0)
      Contact( "Data_ADMIN_HMI".OKE )
      Move(in := 1, out1 => "Data_Control".AUTO."Auto.Mode2_Mode1".Step_ParkingCar)
   END_RUNG
   RUNG wire#powerrail
      { S7_Templates := "SrcType := Int" } EQ_Contact(in1 := "Data_Control".AUTO."Auto.Mode2_Mode1".Step_ParkingCar, in2 := 1)
      { S7_Templates := "SrcType := Int" } NE_Contact(in1 := "Data_Control".Elevator.FloorAddressControlNumber_Check, in2 := 0)
      I_Contact( "Data_Control".TableRotation.Running )
      I_Contact( "Data_Control".Elevator.Running )
      I_Contact( "Data_Control".HookPallet.Running )
      Contact( "Data_Control".Elevator.Done )
      Contact( "Data_Control".HookPallet.Done )
      S_Coil( "Data_Control"."Auto.ACTION".TableRotation_2 )
      Move(in := 2, out1 => "Data_Control".AUTO."Auto.Mode2_Mode1".Step_ParkingCar)
   END_RUNG
   RUNG wire#powerrail
      { S7_Templates := "SrcType := Int" } EQ_Contact(in1 := "Data_Control".AUTO."Auto.Mode2_Mode1".Step_ParkingCar, in2 := 2)
      Contact( "Data_Control".START )
      wire#w1
      { S7_Templates := "SrcType := Int" } EQ_Contact(in1 := "Data_Control".POSITION.POSITIONumber, in2 := 201)
      wire#w2
      Contact( "Data_Control".POSITION."201_C" )
      R_Coil( "Data_Control".POSITION.Parking_Get )
      Move(in := 3, out1 => "Data_Control".AUTO."Auto.Mode2_Mode1".Step_ParkingCar)
   END_RUNG
   RUNG wire#w2
      I_Contact( "Data_Control".POSITION."201_C" )
      S_Coil( "Data_Control".POSITION.Parking_Get )
      Move(in := 3, out1 => "Data_Control".AUTO."Auto.Mode2_Mode1".Step_ParkingCar)
   END_RUNG
   RUNG wire#w1
      { S7_Templates := "SrcType := Int" } EQ_Contact(in1 := "Data_Control".POSITION.POSITIONumber, in2 := 202)
      wire#w3
      Contact( "Data_Control".POSITION."202_C" )
      R_Coil( "Data_Control".POSITION.Parking_Get )
      Move(in := 3, out1 => "Data_Control".AUTO."Auto.Mode2_Mode1".Step_ParkingCar)
   END_RUNG
   RUNG wire#w3
      I_Contact( "Data_Control".POSITION."202_C" )
      S_Coil( "Data_Control".POSITION.Parking_Get )
      Move(in := 3, out1 => "Data_Control".AUTO."Auto.Mode2_Mode1".Step_ParkingCar)
   END_RUNG
   // the same network as SCL:
   IF ("Data_Control".AUTO."Auto.Mode2_Mode1".Step_ParkingCar = 0) AND ("Data_Control".POSITION.POSITIONumber <> 0) AND "Data_ADMIN_HMI".OKE THEN
       "Data_Control".AUTO."Auto.Mode2_Mode1".Step_ParkingCar := 1;
   END_IF;
   IF ("Data_Control".AUTO."Auto.Mode2_Mode1".Step_ParkingCar = 1) AND ("Data_Control".Elevator.FloorAddressControlNumber_Check <> 0) AND NOT "Data_Control".TableRotation.Running AND NOT "Data_Control".Elevator.Running AND NOT "Data_Control".HookPallet.Running AND "Data_Control".Elevator.Done AND "Data_Control".HookPallet.Done THEN
       "Data_Control"."Auto.ACTION".TableRotation_2 := TRUE;
       "Data_Control".AUTO."Auto.Mode2_Mode1".Step_ParkingCar := 2;
   END_IF;
   #_w1 := ("Data_Control".AUTO."Auto.Mode2_Mode1".Step_ParkingCar = 2) AND "Data_Control".START;
   #_w2 := #_w1 AND ("Data_Control".POSITION.POSITIONumber = 201);
   IF #_w2 AND "Data_Control".POSITION."201_C" THEN
       "Data_Control".POSITION.Parking_Get := FALSE;
       "Data_Control".AUTO."Auto.Mode2_Mode1".Step_ParkingCar := 3;
   END_IF;
   IF #_w2 AND NOT "Data_Control".POSITION."201_C" THEN
       "Data_Control".POSITION.Parking_Get := TRUE;
       "Data_Control".AUTO."Auto.Mode2_Mode1".Step_ParkingCar := 3;
   END_IF;
   #_w3 := #_w1 AND ("Data_Control".POSITION.POSITIONumber = 202);
   IF #_w3 AND "Data_Control".POSITION."202_C" THEN
       "Data_Control".POSITION.Parking_Get := FALSE;
       "Data_Control".AUTO."Auto.Mode2_Mode1".Step_ParkingCar := 3;
   END_IF;
   IF #_w3 AND NOT "Data_Control".POSITION."202_C" THEN
       "Data_Control".POSITION.Parking_Get := TRUE;
       "Data_Control".AUTO."Auto.Mode2_Mode1".Step_ParkingCar := 3;
   END_IF;
END_REGION

REGION Network 2
   // Up
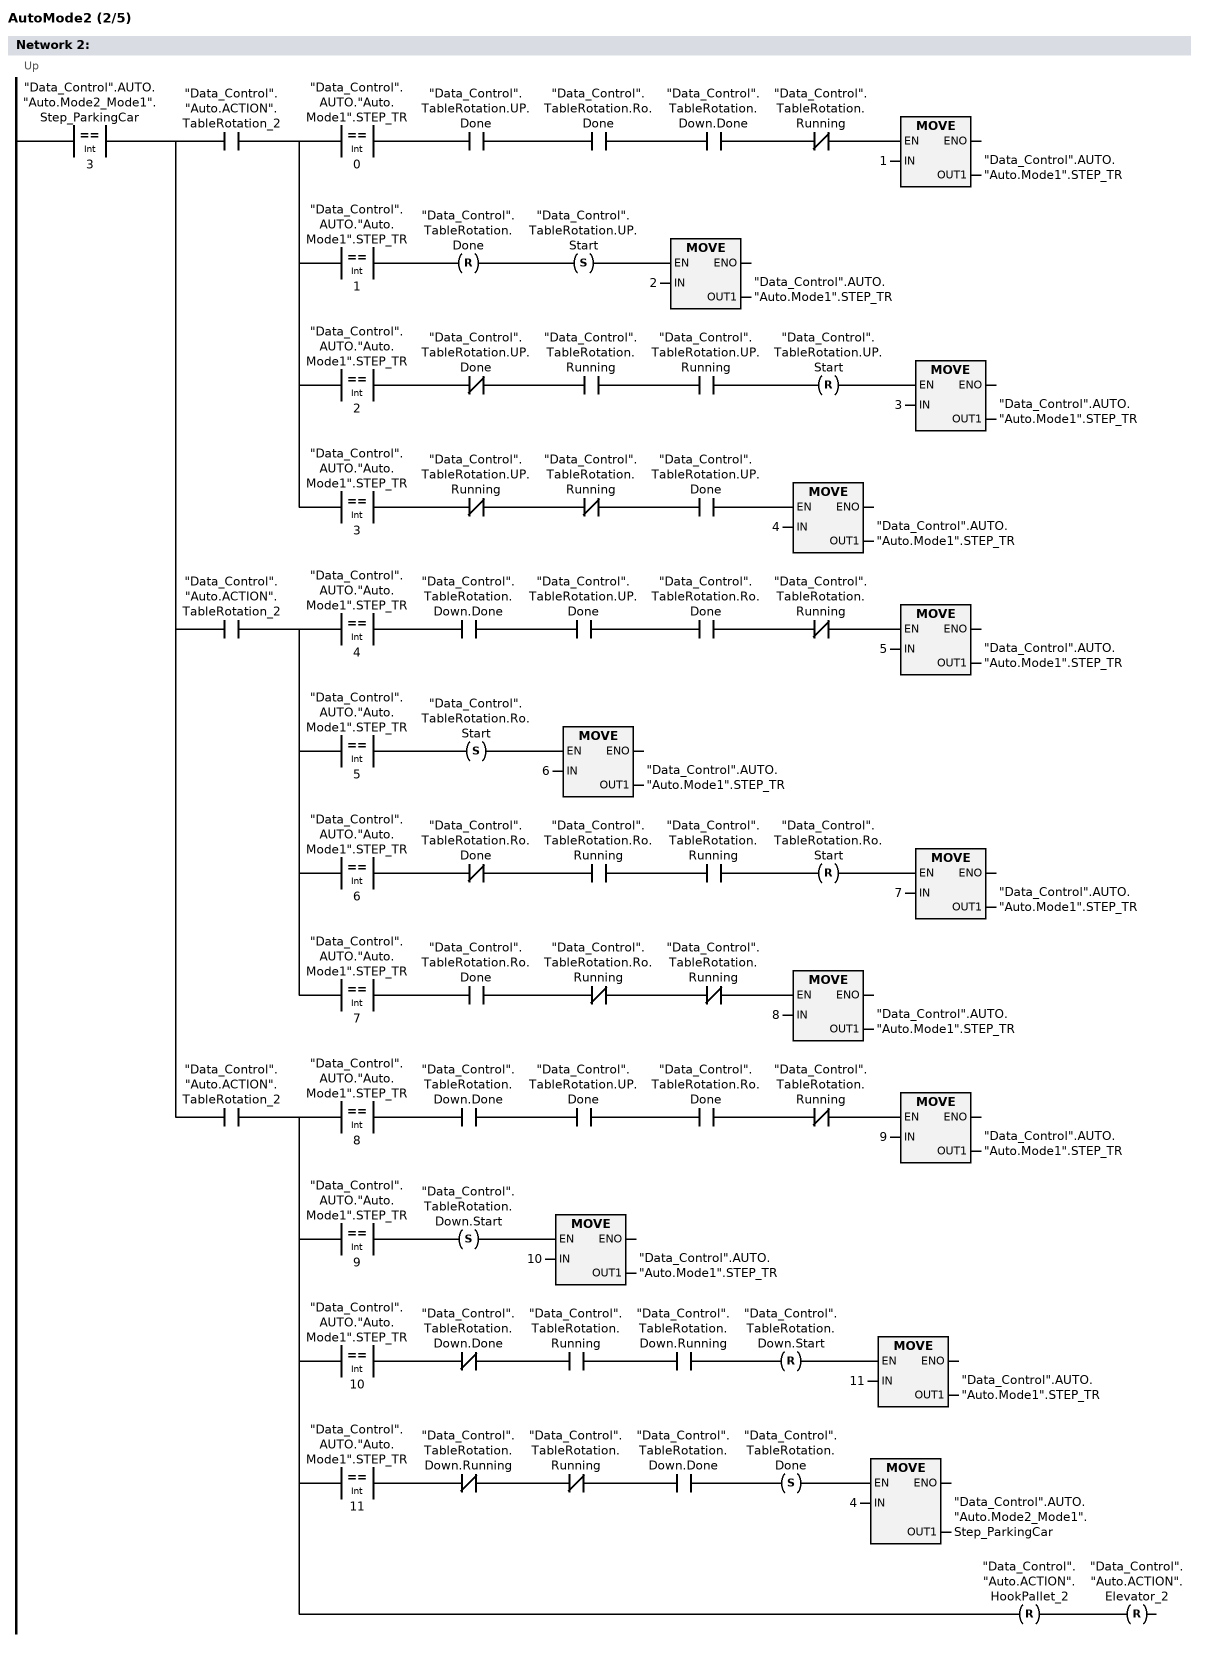
   RUNG wire#powerrail
      { S7_Templates := "SrcType := Int" } EQ_Contact(in1 := "Data_Control".AUTO."Auto.Mode2_Mode1".Step_ParkingCar, in2 := 3)
      wire#w1
      Contact( "Data_Control"."Auto.ACTION".TableRotation_2 )
      wire#w2
      { S7_Templates := "SrcType := Int" } EQ_Contact(in1 := "Data_Control".AUTO."Auto.Mode1".STEP_TR, in2 := 0)
      Contact( "Data_Control".TableRotation.UP.Done )
      Contact( "Data_Control".TableRotation.Ro.Done )
      Contact( "Data_Control".TableRotation.Down.Done )
      I_Contact( "Data_Control".TableRotation.Running )
      Move(in := 1, out1 => "Data_Control".AUTO."Auto.Mode1".STEP_TR)
   END_RUNG
   RUNG wire#w2
      { S7_Templates := "SrcType := Int" } EQ_Contact(in1 := "Data_Control".AUTO."Auto.Mode1".STEP_TR, in2 := 1)
      R_Coil( "Data_Control".TableRotation.Done )
      S_Coil( "Data_Control".TableRotation.UP.Start )
      Move(in := 2, out1 => "Data_Control".AUTO."Auto.Mode1".STEP_TR)
   END_RUNG
   RUNG wire#w2
      { S7_Templates := "SrcType := Int" } EQ_Contact(in1 := "Data_Control".AUTO."Auto.Mode1".STEP_TR, in2 := 2)
      I_Contact( "Data_Control".TableRotation.UP.Done )
      Contact( "Data_Control".TableRotation.Running )
      Contact( "Data_Control".TableRotation.UP.Running )
      R_Coil( "Data_Control".TableRotation.UP.Start )
      Move(in := 3, out1 => "Data_Control".AUTO."Auto.Mode1".STEP_TR)
   END_RUNG
   RUNG wire#w2
      { S7_Templates := "SrcType := Int" } EQ_Contact(in1 := "Data_Control".AUTO."Auto.Mode1".STEP_TR, in2 := 3)
      I_Contact( "Data_Control".TableRotation.UP.Running )
      I_Contact( "Data_Control".TableRotation.Running )
      Contact( "Data_Control".TableRotation.UP.Done )
      Move(in := 4, out1 => "Data_Control".AUTO."Auto.Mode1".STEP_TR)
   END_RUNG
   RUNG wire#w1
      Contact( "Data_Control"."Auto.ACTION".TableRotation_2 )
      wire#w3
      { S7_Templates := "SrcType := Int" } EQ_Contact(in1 := "Data_Control".AUTO."Auto.Mode1".STEP_TR, in2 := 4)
      Contact( "Data_Control".TableRotation.Down.Done )
      Contact( "Data_Control".TableRotation.UP.Done )
      Contact( "Data_Control".TableRotation.Ro.Done )
      I_Contact( "Data_Control".TableRotation.Running )
      Move(in := 5, out1 => "Data_Control".AUTO."Auto.Mode1".STEP_TR)
   END_RUNG
   RUNG wire#w3
      { S7_Templates := "SrcType := Int" } EQ_Contact(in1 := "Data_Control".AUTO."Auto.Mode1".STEP_TR, in2 := 5)
      S_Coil( "Data_Control".TableRotation.Ro.Start )
      Move(in := 6, out1 => "Data_Control".AUTO."Auto.Mode1".STEP_TR)
   END_RUNG
   RUNG wire#w3
      { S7_Templates := "SrcType := Int" } EQ_Contact(in1 := "Data_Control".AUTO."Auto.Mode1".STEP_TR, in2 := 6)
      I_Contact( "Data_Control".TableRotation.Ro.Done )
      Contact( "Data_Control".TableRotation.Ro.Running )
      Contact( "Data_Control".TableRotation.Running )
      R_Coil( "Data_Control".TableRotation.Ro.Start )
      Move(in := 7, out1 => "Data_Control".AUTO."Auto.Mode1".STEP_TR)
   END_RUNG
   RUNG wire#w3
      { S7_Templates := "SrcType := Int" } EQ_Contact(in1 := "Data_Control".AUTO."Auto.Mode1".STEP_TR, in2 := 7)
      Contact( "Data_Control".TableRotation.Ro.Done )
      I_Contact( "Data_Control".TableRotation.Ro.Running )
      I_Contact( "Data_Control".TableRotation.Running )
      Move(in := 8, out1 => "Data_Control".AUTO."Auto.Mode1".STEP_TR)
   END_RUNG
   RUNG wire#w1
      Contact( "Data_Control"."Auto.ACTION".TableRotation_2 )
      wire#w4
      { S7_Templates := "SrcType := Int" } EQ_Contact(in1 := "Data_Control".AUTO."Auto.Mode1".STEP_TR, in2 := 8)
      Contact( "Data_Control".TableRotation.Down.Done )
      Contact( "Data_Control".TableRotation.UP.Done )
      Contact( "Data_Control".TableRotation.Ro.Done )
      I_Contact( "Data_Control".TableRotation.Running )
      Move(in := 9, out1 => "Data_Control".AUTO."Auto.Mode1".STEP_TR)
   END_RUNG
   RUNG wire#w4
      { S7_Templates := "SrcType := Int" } EQ_Contact(in1 := "Data_Control".AUTO."Auto.Mode1".STEP_TR, in2 := 9)
      S_Coil( "Data_Control".TableRotation.Down.Start )
      Move(in := 10, out1 => "Data_Control".AUTO."Auto.Mode1".STEP_TR)
   END_RUNG
   RUNG wire#w4
      { S7_Templates := "SrcType := Int" } EQ_Contact(in1 := "Data_Control".AUTO."Auto.Mode1".STEP_TR, in2 := 10)
      I_Contact( "Data_Control".TableRotation.Down.Done )
      Contact( "Data_Control".TableRotation.Running )
      Contact( "Data_Control".TableRotation.Down.Running )
      R_Coil( "Data_Control".TableRotation.Down.Start )
      Move(in := 11, out1 => "Data_Control".AUTO."Auto.Mode1".STEP_TR)
   END_RUNG
   RUNG wire#w4
      { S7_Templates := "SrcType := Int" } EQ_Contact(in1 := "Data_Control".AUTO."Auto.Mode1".STEP_TR, in2 := 11)
      I_Contact( "Data_Control".TableRotation.Down.Running )
      I_Contact( "Data_Control".TableRotation.Running )
      Contact( "Data_Control".TableRotation.Down.Done )
      S_Coil( "Data_Control".TableRotation.Done )
      Move(in := 4, out1 => "Data_Control".AUTO."Auto.Mode2_Mode1".Step_ParkingCar)
   END_RUNG
   RUNG wire#w4
      R_Coil( "Data_Control"."Auto.ACTION".HookPallet_2 )
      R_Coil( "Data_Control"."Auto.ACTION".Elevator_2 )
   END_RUNG
   // the same network as SCL:
   #_w1 := "Data_Control".AUTO."Auto.Mode2_Mode1".Step_ParkingCar = 3;
   #_w2 := #_w1 AND "Data_Control"."Auto.ACTION".TableRotation_2;
   IF #_w2 AND ("Data_Control".AUTO."Auto.Mode1".STEP_TR = 0) AND "Data_Control".TableRotation.UP.Done AND "Data_Control".TableRotation.Ro.Done AND "Data_Control".TableRotation.Down.Done AND NOT "Data_Control".TableRotation.Running THEN
       "Data_Control".AUTO."Auto.Mode1".STEP_TR := 1;
   END_IF;
   IF #_w2 AND ("Data_Control".AUTO."Auto.Mode1".STEP_TR = 1) THEN
       "Data_Control".TableRotation.Done := FALSE;
       "Data_Control".TableRotation.UP.Start := TRUE;
       "Data_Control".AUTO."Auto.Mode1".STEP_TR := 2;
   END_IF;
   IF #_w2 AND ("Data_Control".AUTO."Auto.Mode1".STEP_TR = 2) AND NOT "Data_Control".TableRotation.UP.Done AND "Data_Control".TableRotation.Running AND "Data_Control".TableRotation.UP.Running THEN
       "Data_Control".TableRotation.UP.Start := FALSE;
       "Data_Control".AUTO."Auto.Mode1".STEP_TR := 3;
   END_IF;
   IF #_w2 AND ("Data_Control".AUTO."Auto.Mode1".STEP_TR = 3) AND NOT "Data_Control".TableRotation.UP.Running AND NOT "Data_Control".TableRotation.Running AND "Data_Control".TableRotation.UP.Done THEN
       "Data_Control".AUTO."Auto.Mode1".STEP_TR := 4;
   END_IF;
   #_w3 := #_w1 AND "Data_Control"."Auto.ACTION".TableRotation_2;
   IF #_w3 AND ("Data_Control".AUTO."Auto.Mode1".STEP_TR = 4) AND "Data_Control".TableRotation.Down.Done AND "Data_Control".TableRotation.UP.Done AND "Data_Control".TableRotation.Ro.Done AND NOT "Data_Control".TableRotation.Running THEN
       "Data_Control".AUTO."Auto.Mode1".STEP_TR := 5;
   END_IF;
   IF #_w3 AND ("Data_Control".AUTO."Auto.Mode1".STEP_TR = 5) THEN
       "Data_Control".TableRotation.Ro.Start := TRUE;
       "Data_Control".AUTO."Auto.Mode1".STEP_TR := 6;
   END_IF;
   IF #_w3 AND ("Data_Control".AUTO."Auto.Mode1".STEP_TR = 6) AND NOT "Data_Control".TableRotation.Ro.Done AND "Data_Control".TableRotation.Ro.Running AND "Data_Control".TableRotation.Running THEN
       "Data_Control".TableRotation.Ro.Start := FALSE;
       "Data_Control".AUTO."Auto.Mode1".STEP_TR := 7;
   END_IF;
   IF #_w3 AND ("Data_Control".AUTO."Auto.Mode1".STEP_TR = 7) AND "Data_Control".TableRotation.Ro.Done AND NOT "Data_Control".TableRotation.Ro.Running AND NOT "Data_Control".TableRotation.Running THEN
       "Data_Control".AUTO."Auto.Mode1".STEP_TR := 8;
   END_IF;
   #_w4 := #_w1 AND "Data_Control"."Auto.ACTION".TableRotation_2;
   IF #_w4 AND ("Data_Control".AUTO."Auto.Mode1".STEP_TR = 8) AND "Data_Control".TableRotation.Down.Done AND "Data_Control".TableRotation.UP.Done AND "Data_Control".TableRotation.Ro.Done AND NOT "Data_Control".TableRotation.Running THEN
       "Data_Control".AUTO."Auto.Mode1".STEP_TR := 9;
   END_IF;
   IF #_w4 AND ("Data_Control".AUTO."Auto.Mode1".STEP_TR = 9) THEN
       "Data_Control".TableRotation.Down.Start := TRUE;
       "Data_Control".AUTO."Auto.Mode1".STEP_TR := 10;
   END_IF;
   IF #_w4 AND ("Data_Control".AUTO."Auto.Mode1".STEP_TR = 10) AND NOT "Data_Control".TableRotation.Down.Done AND "Data_Control".TableRotation.Running AND "Data_Control".TableRotation.Down.Running THEN
       "Data_Control".TableRotation.Down.Start := FALSE;
       "Data_Control".AUTO."Auto.Mode1".STEP_TR := 11;
   END_IF;
   IF #_w4 AND ("Data_Control".AUTO."Auto.Mode1".STEP_TR = 11) AND NOT "Data_Control".TableRotation.Down.Running AND NOT "Data_Control".TableRotation.Running AND "Data_Control".TableRotation.Down.Done THEN
       "Data_Control".TableRotation.Done := TRUE;
       "Data_Control".AUTO."Auto.Mode2_Mode1".Step_ParkingCar := 4;
   END_IF;
   IF #_w4 THEN
       "Data_Control"."Auto.ACTION".HookPallet_2 := FALSE;
       "Data_Control"."Auto.ACTION".Elevator_2 := FALSE;
   END_IF;
END_REGION

REGION Network 3
   // Ro
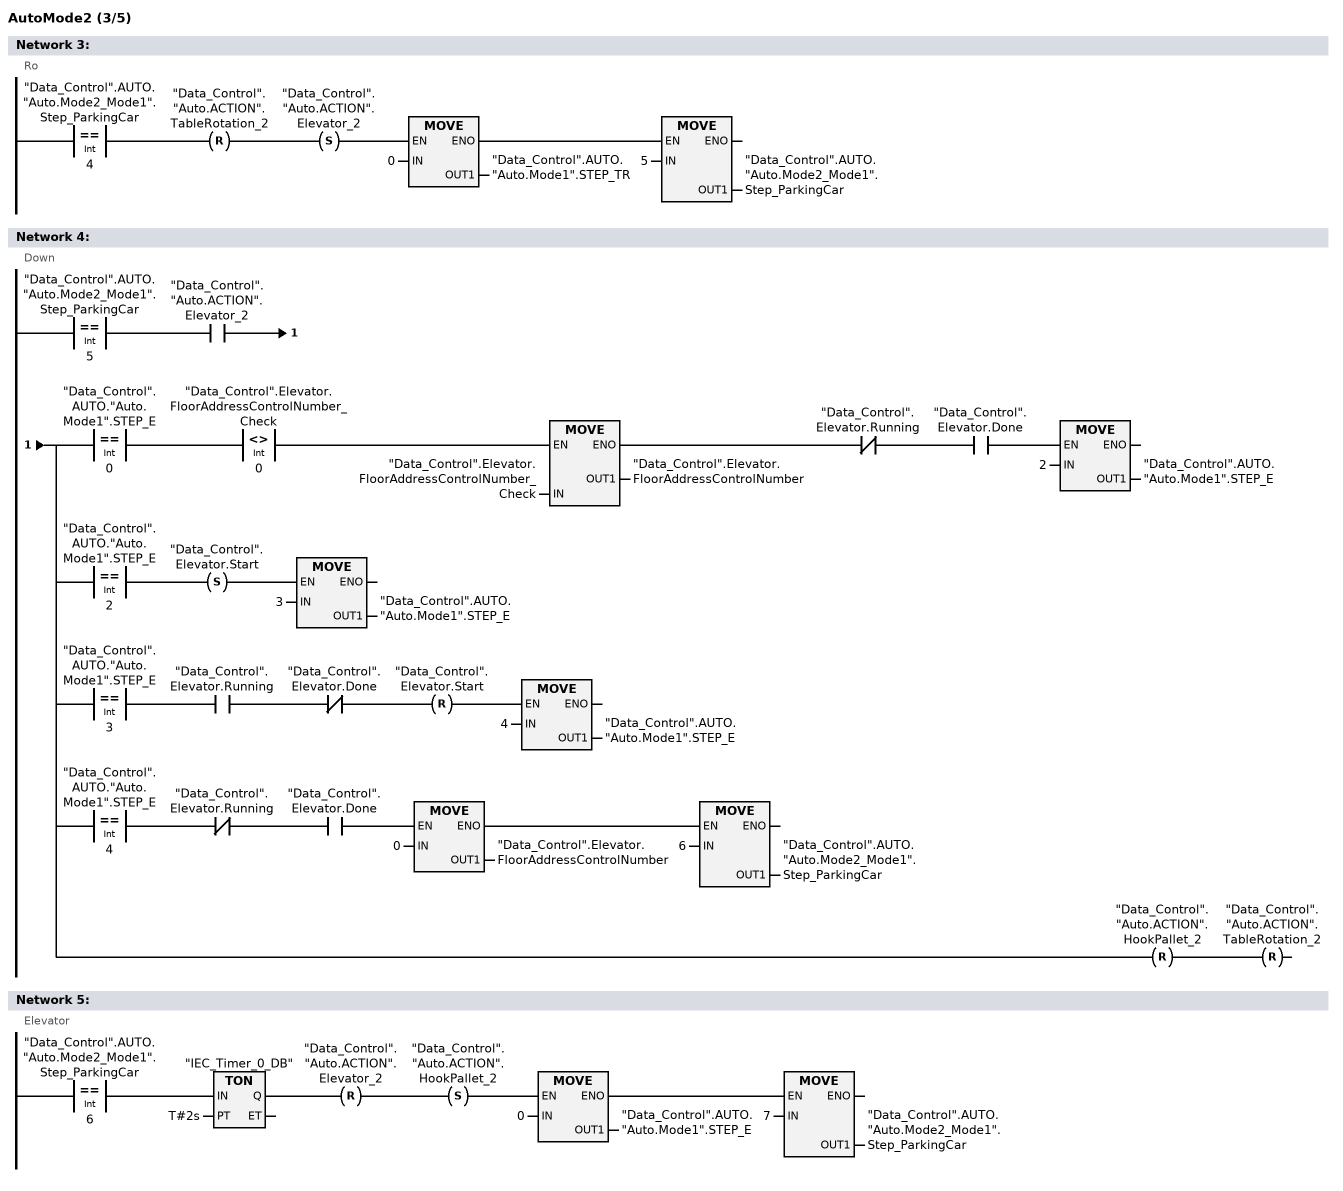
   RUNG wire#powerrail
      { S7_Templates := "SrcType := Int" } EQ_Contact(in1 := "Data_Control".AUTO."Auto.Mode2_Mode1".Step_ParkingCar, in2 := 4)
      R_Coil( "Data_Control"."Auto.ACTION".TableRotation_2 )
      S_Coil( "Data_Control"."Auto.ACTION".Elevator_2 )
      Move(in := 0, out1 => "Data_Control".AUTO."Auto.Mode1".STEP_TR)
      Move(in := 5, out1 => "Data_Control".AUTO."Auto.Mode2_Mode1".Step_ParkingCar)
   END_RUNG
   // the same network as SCL:
   IF "Data_Control".AUTO."Auto.Mode2_Mode1".Step_ParkingCar = 4 THEN
       "Data_Control"."Auto.ACTION".TableRotation_2 := FALSE;
       "Data_Control"."Auto.ACTION".Elevator_2 := TRUE;
       "Data_Control".AUTO."Auto.Mode1".STEP_TR := 0;
       "Data_Control".AUTO."Auto.Mode2_Mode1".Step_ParkingCar := 5;
   END_IF;
END_REGION

REGION Network 4
   // Down
   RUNG wire#powerrail
      { S7_Templates := "SrcType := Int" } EQ_Contact(in1 := "Data_Control".AUTO."Auto.Mode2_Mode1".Step_ParkingCar, in2 := 5)
      Contact( "Data_Control"."Auto.ACTION".Elevator_2 )
      wire#w1
      { S7_Templates := "SrcType := Int" } EQ_Contact(in1 := "Data_Control".AUTO."Auto.Mode1".STEP_E, in2 := 0)
      { S7_Templates := "SrcType := Int" } NE_Contact(in1 := "Data_Control".Elevator.FloorAddressControlNumber_Check, in2 := 0)
      Move(in := "Data_Control".Elevator.FloorAddressControlNumber_Check, out1 => "Data_Control".Elevator.FloorAddressControlNumber)
      I_Contact( "Data_Control".Elevator.Running )
      Contact( "Data_Control".Elevator.Done )
      Move(in := 2, out1 => "Data_Control".AUTO."Auto.Mode1".STEP_E)
   END_RUNG
   RUNG wire#w1
      { S7_Templates := "SrcType := Int" } EQ_Contact(in1 := "Data_Control".AUTO."Auto.Mode1".STEP_E, in2 := 2)
      S_Coil( "Data_Control".Elevator.Start )
      Move(in := 3, out1 => "Data_Control".AUTO."Auto.Mode1".STEP_E)
   END_RUNG
   RUNG wire#w1
      { S7_Templates := "SrcType := Int" } EQ_Contact(in1 := "Data_Control".AUTO."Auto.Mode1".STEP_E, in2 := 3)
      Contact( "Data_Control".Elevator.Running )
      I_Contact( "Data_Control".Elevator.Done )
      R_Coil( "Data_Control".Elevator.Start )
      Move(in := 4, out1 => "Data_Control".AUTO."Auto.Mode1".STEP_E)
   END_RUNG
   RUNG wire#w1
      { S7_Templates := "SrcType := Int" } EQ_Contact(in1 := "Data_Control".AUTO."Auto.Mode1".STEP_E, in2 := 4)
      I_Contact( "Data_Control".Elevator.Running )
      Contact( "Data_Control".Elevator.Done )
      Move(in := 0, out1 => "Data_Control".Elevator.FloorAddressControlNumber)
      Move(in := 6, out1 => "Data_Control".AUTO."Auto.Mode2_Mode1".Step_ParkingCar)
   END_RUNG
   RUNG wire#w1
      R_Coil( "Data_Control"."Auto.ACTION".HookPallet_2 )
      R_Coil( "Data_Control"."Auto.ACTION".TableRotation_2 )
   END_RUNG
   // the same network as SCL:
   #_w1 := ("Data_Control".AUTO."Auto.Mode2_Mode1".Step_ParkingCar = 5) AND "Data_Control"."Auto.ACTION".Elevator_2;
   #_w2 := #_w1 AND ("Data_Control".AUTO."Auto.Mode1".STEP_E = 0) AND ("Data_Control".Elevator.FloorAddressControlNumber_Check <> 0);
   IF #_w2 THEN
       "Data_Control".Elevator.FloorAddressControlNumber := "Data_Control".Elevator.FloorAddressControlNumber_Check;
   END_IF;
   IF #_w2 AND NOT "Data_Control".Elevator.Running AND "Data_Control".Elevator.Done THEN
       "Data_Control".AUTO."Auto.Mode1".STEP_E := 2;
   END_IF;
   IF #_w1 AND ("Data_Control".AUTO."Auto.Mode1".STEP_E = 2) THEN
       "Data_Control".Elevator.Start := TRUE;
       "Data_Control".AUTO."Auto.Mode1".STEP_E := 3;
   END_IF;
   IF #_w1 AND ("Data_Control".AUTO."Auto.Mode1".STEP_E = 3) AND "Data_Control".Elevator.Running AND NOT "Data_Control".Elevator.Done THEN
       "Data_Control".Elevator.Start := FALSE;
       "Data_Control".AUTO."Auto.Mode1".STEP_E := 4;
   END_IF;
   IF #_w1 AND ("Data_Control".AUTO."Auto.Mode1".STEP_E = 4) AND NOT "Data_Control".Elevator.Running AND "Data_Control".Elevator.Done THEN
       "Data_Control".Elevator.FloorAddressControlNumber := 0;
       "Data_Control".AUTO."Auto.Mode2_Mode1".Step_ParkingCar := 6;
   END_IF;
   IF #_w1 THEN
       "Data_Control"."Auto.ACTION".HookPallet_2 := FALSE;
       "Data_Control"."Auto.ACTION".TableRotation_2 := FALSE;
   END_IF;
END_REGION

REGION Network 5
   // Elevator
   "IEC_Timer_0_DB".TON(IN := "Data_Control".AUTO."Auto.Mode2_Mode1".Step_ParkingCar = 6, PT := T#2s);
   IF "IEC_Timer_0_DB".Q THEN
       "Data_Control"."Auto.ACTION".Elevator_2 := FALSE;
       "Data_Control"."Auto.ACTION".HookPallet_2 := TRUE;
       "Data_Control".AUTO."Auto.Mode1".STEP_E := 0;
       "Data_Control".AUTO."Auto.Mode2_Mode1".Step_ParkingCar := 7;
   END_IF;
END_REGION

REGION Network 6
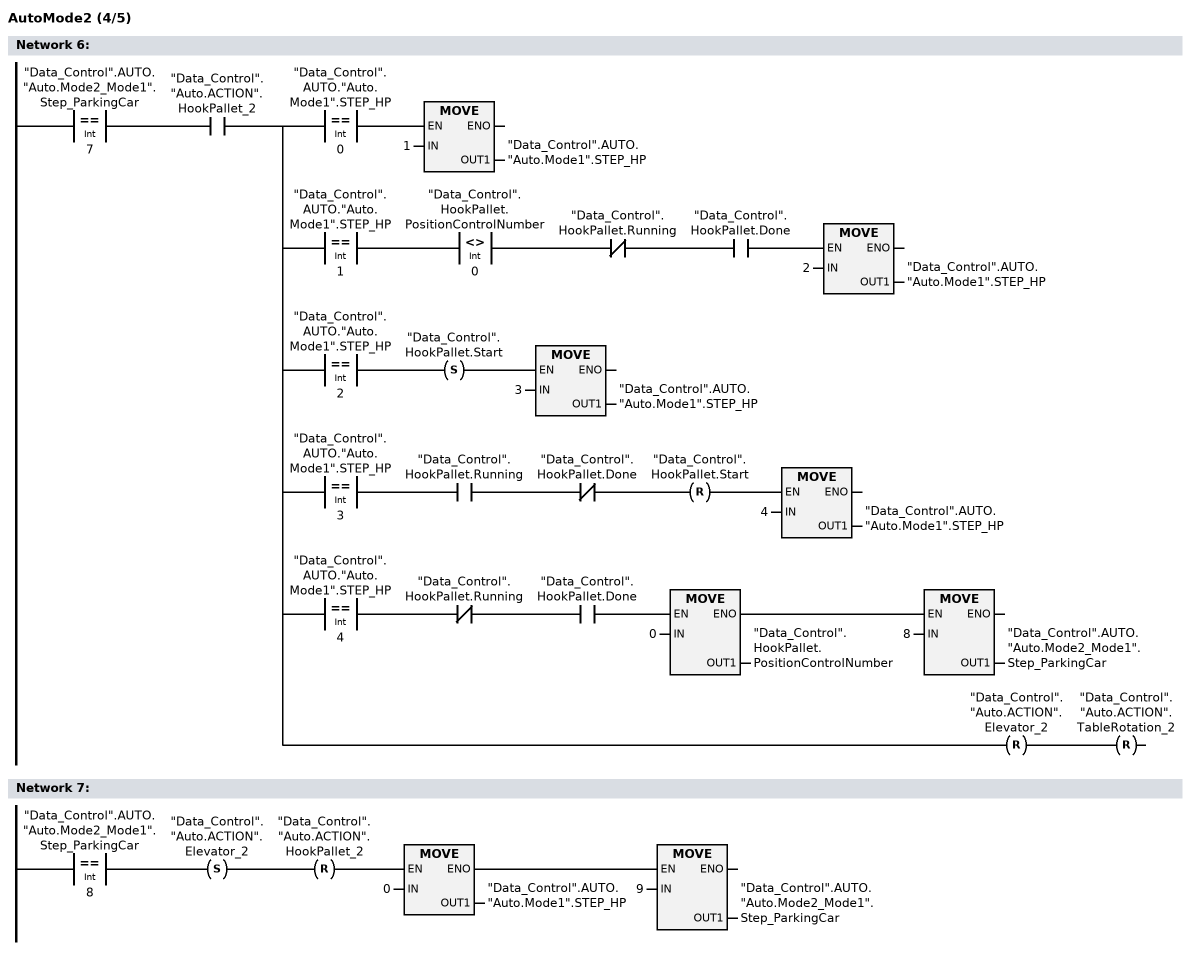
   RUNG wire#powerrail
      { S7_Templates := "SrcType := Int" } EQ_Contact(in1 := "Data_Control".AUTO."Auto.Mode2_Mode1".Step_ParkingCar, in2 := 7)
      Contact( "Data_Control"."Auto.ACTION".HookPallet_2 )
      wire#w1
      { S7_Templates := "SrcType := Int" } EQ_Contact(in1 := "Data_Control".AUTO."Auto.Mode1".STEP_HP, in2 := 0)
      Move(in := 1, out1 => "Data_Control".AUTO."Auto.Mode1".STEP_HP)
   END_RUNG
   RUNG wire#w1
      { S7_Templates := "SrcType := Int" } EQ_Contact(in1 := "Data_Control".AUTO."Auto.Mode1".STEP_HP, in2 := 1)
      { S7_Templates := "SrcType := Int" } NE_Contact(in1 := "Data_Control".HookPallet.PositionControlNumber, in2 := 0)
      I_Contact( "Data_Control".HookPallet.Running )
      Contact( "Data_Control".HookPallet.Done )
      Move(in := 2, out1 => "Data_Control".AUTO."Auto.Mode1".STEP_HP)
   END_RUNG
   RUNG wire#w1
      { S7_Templates := "SrcType := Int" } EQ_Contact(in1 := "Data_Control".AUTO."Auto.Mode1".STEP_HP, in2 := 2)
      S_Coil( "Data_Control".HookPallet.Start )
      Move(in := 3, out1 => "Data_Control".AUTO."Auto.Mode1".STEP_HP)
   END_RUNG
   RUNG wire#w1
      { S7_Templates := "SrcType := Int" } EQ_Contact(in1 := "Data_Control".AUTO."Auto.Mode1".STEP_HP, in2 := 3)
      Contact( "Data_Control".HookPallet.Running )
      I_Contact( "Data_Control".HookPallet.Done )
      R_Coil( "Data_Control".HookPallet.Start )
      Move(in := 4, out1 => "Data_Control".AUTO."Auto.Mode1".STEP_HP)
   END_RUNG
   RUNG wire#w1
      { S7_Templates := "SrcType := Int" } EQ_Contact(in1 := "Data_Control".AUTO."Auto.Mode1".STEP_HP, in2 := 4)
      I_Contact( "Data_Control".HookPallet.Running )
      Contact( "Data_Control".HookPallet.Done )
      Move(in := 0, out1 => "Data_Control".HookPallet.PositionControlNumber)
      Move(in := 8, out1 => "Data_Control".AUTO."Auto.Mode2_Mode1".Step_ParkingCar)
   END_RUNG
   RUNG wire#w1
      R_Coil( "Data_Control"."Auto.ACTION".Elevator_2 )
      R_Coil( "Data_Control"."Auto.ACTION".TableRotation_2 )
   END_RUNG
   // the same network as SCL:
   #_w1 := ("Data_Control".AUTO."Auto.Mode2_Mode1".Step_ParkingCar = 7) AND "Data_Control"."Auto.ACTION".HookPallet_2;
   IF #_w1 AND ("Data_Control".AUTO."Auto.Mode1".STEP_HP = 0) THEN
       "Data_Control".AUTO."Auto.Mode1".STEP_HP := 1;
   END_IF;
   IF #_w1 AND ("Data_Control".AUTO."Auto.Mode1".STEP_HP = 1) AND ("Data_Control".HookPallet.PositionControlNumber <> 0) AND NOT "Data_Control".HookPallet.Running AND "Data_Control".HookPallet.Done THEN
       "Data_Control".AUTO."Auto.Mode1".STEP_HP := 2;
   END_IF;
   IF #_w1 AND ("Data_Control".AUTO."Auto.Mode1".STEP_HP = 2) THEN
       "Data_Control".HookPallet.Start := TRUE;
       "Data_Control".AUTO."Auto.Mode1".STEP_HP := 3;
   END_IF;
   IF #_w1 AND ("Data_Control".AUTO."Auto.Mode1".STEP_HP = 3) AND "Data_Control".HookPallet.Running AND NOT "Data_Control".HookPallet.Done THEN
       "Data_Control".HookPallet.Start := FALSE;
       "Data_Control".AUTO."Auto.Mode1".STEP_HP := 4;
   END_IF;
   IF #_w1 AND ("Data_Control".AUTO."Auto.Mode1".STEP_HP = 4) AND NOT "Data_Control".HookPallet.Running AND "Data_Control".HookPallet.Done THEN
       "Data_Control".HookPallet.PositionControlNumber := 0;
       "Data_Control".AUTO."Auto.Mode2_Mode1".Step_ParkingCar := 8;
   END_IF;
   IF #_w1 THEN
       "Data_Control"."Auto.ACTION".Elevator_2 := FALSE;
       "Data_Control"."Auto.ACTION".TableRotation_2 := FALSE;
   END_IF;
END_REGION

REGION Network 7
   RUNG wire#powerrail
      { S7_Templates := "SrcType := Int" } EQ_Contact(in1 := "Data_Control".AUTO."Auto.Mode2_Mode1".Step_ParkingCar, in2 := 8)
      S_Coil( "Data_Control"."Auto.ACTION".Elevator_2 )
      R_Coil( "Data_Control"."Auto.ACTION".HookPallet_2 )
      Move(in := 0, out1 => "Data_Control".AUTO."Auto.Mode1".STEP_HP)
      Move(in := 9, out1 => "Data_Control".AUTO."Auto.Mode2_Mode1".Step_ParkingCar)
   END_RUNG
   // the same network as SCL:
   IF "Data_Control".AUTO."Auto.Mode2_Mode1".Step_ParkingCar = 8 THEN
       "Data_Control"."Auto.ACTION".Elevator_2 := TRUE;
       "Data_Control"."Auto.ACTION".HookPallet_2 := FALSE;
       "Data_Control".AUTO."Auto.Mode1".STEP_HP := 0;
       "Data_Control".AUTO."Auto.Mode2_Mode1".Step_ParkingCar := 9;
   END_IF;
END_REGION

REGION Network 8
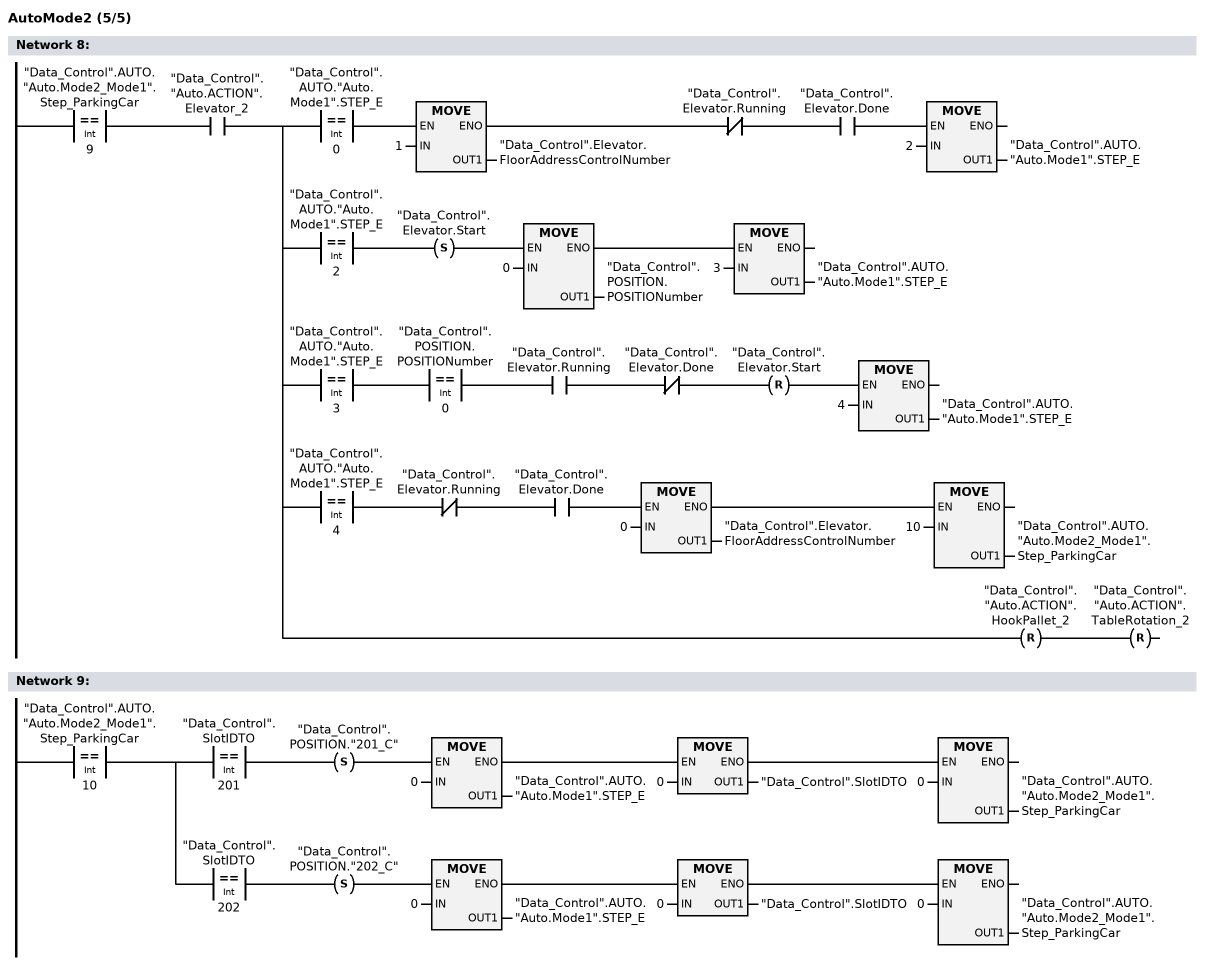
   RUNG wire#powerrail
      { S7_Templates := "SrcType := Int" } EQ_Contact(in1 := "Data_Control".AUTO."Auto.Mode2_Mode1".Step_ParkingCar, in2 := 9)
      Contact( "Data_Control"."Auto.ACTION".Elevator_2 )
      wire#w1
      { S7_Templates := "SrcType := Int" } EQ_Contact(in1 := "Data_Control".AUTO."Auto.Mode1".STEP_E, in2 := 0)
      Move(in := 1, out1 => "Data_Control".Elevator.FloorAddressControlNumber)
      I_Contact( "Data_Control".Elevator.Running )
      Contact( "Data_Control".Elevator.Done )
      Move(in := 2, out1 => "Data_Control".AUTO."Auto.Mode1".STEP_E)
   END_RUNG
   RUNG wire#w1
      { S7_Templates := "SrcType := Int" } EQ_Contact(in1 := "Data_Control".AUTO."Auto.Mode1".STEP_E, in2 := 2)
      S_Coil( "Data_Control".Elevator.Start )
      Move(in := 0, out1 => "Data_Control".POSITION.POSITIONumber)
      Move(in := 3, out1 => "Data_Control".AUTO."Auto.Mode1".STEP_E)
   END_RUNG
   RUNG wire#w1
      { S7_Templates := "SrcType := Int" } EQ_Contact(in1 := "Data_Control".AUTO."Auto.Mode1".STEP_E, in2 := 3)
      { S7_Templates := "SrcType := Int" } EQ_Contact(in1 := "Data_Control".POSITION.POSITIONumber, in2 := 0)
      Contact( "Data_Control".Elevator.Running )
      I_Contact( "Data_Control".Elevator.Done )
      R_Coil( "Data_Control".Elevator.Start )
      Move(in := 4, out1 => "Data_Control".AUTO."Auto.Mode1".STEP_E)
   END_RUNG
   RUNG wire#w1
      { S7_Templates := "SrcType := Int" } EQ_Contact(in1 := "Data_Control".AUTO."Auto.Mode1".STEP_E, in2 := 4)
      I_Contact( "Data_Control".Elevator.Running )
      Contact( "Data_Control".Elevator.Done )
      Move(in := 0, out1 => "Data_Control".Elevator.FloorAddressControlNumber)
      Move(in := 10, out1 => "Data_Control".AUTO."Auto.Mode2_Mode1".Step_ParkingCar)
   END_RUNG
   RUNG wire#w1
      R_Coil( "Data_Control"."Auto.ACTION".HookPallet_2 )
      R_Coil( "Data_Control"."Auto.ACTION".TableRotation_2 )
   END_RUNG
   // the same network as SCL:
   #_w1 := ("Data_Control".AUTO."Auto.Mode2_Mode1".Step_ParkingCar = 9) AND "Data_Control"."Auto.ACTION".Elevator_2;
   #_w2 := #_w1 AND ("Data_Control".AUTO."Auto.Mode1".STEP_E = 0);
   IF #_w2 THEN "Data_Control".Elevator.FloorAddressControlNumber := 1; END_IF;
   IF #_w2 AND NOT "Data_Control".Elevator.Running AND "Data_Control".Elevator.Done THEN
       "Data_Control".AUTO."Auto.Mode1".STEP_E := 2;
   END_IF;
   IF #_w1 AND ("Data_Control".AUTO."Auto.Mode1".STEP_E = 2) THEN
       "Data_Control".Elevator.Start := TRUE;
       "Data_Control".POSITION.POSITIONumber := 0;
       "Data_Control".AUTO."Auto.Mode1".STEP_E := 3;
   END_IF;
   IF #_w1 AND ("Data_Control".AUTO."Auto.Mode1".STEP_E = 3) AND ("Data_Control".POSITION.POSITIONumber = 0) AND "Data_Control".Elevator.Running AND NOT "Data_Control".Elevator.Done THEN
       "Data_Control".Elevator.Start := FALSE;
       "Data_Control".AUTO."Auto.Mode1".STEP_E := 4;
   END_IF;
   IF #_w1 AND ("Data_Control".AUTO."Auto.Mode1".STEP_E = 4) AND NOT "Data_Control".Elevator.Running AND "Data_Control".Elevator.Done THEN
       "Data_Control".Elevator.FloorAddressControlNumber := 0;
       "Data_Control".AUTO."Auto.Mode2_Mode1".Step_ParkingCar := 10;
   END_IF;
   IF #_w1 THEN
       "Data_Control"."Auto.ACTION".HookPallet_2 := FALSE;
       "Data_Control"."Auto.ACTION".TableRotation_2 := FALSE;
   END_IF;
END_REGION

REGION Network 9
   RUNG wire#powerrail
      { S7_Templates := "SrcType := Int" } EQ_Contact(in1 := "Data_Control".AUTO."Auto.Mode2_Mode1".Step_ParkingCar, in2 := 10)
      wire#w1
      { S7_Templates := "SrcType := Int" } EQ_Contact(in1 := "Data_Control".SlotIDTO, in2 := 201)
      S_Coil( "Data_Control".POSITION."201_C" )
      Move(in := 0, out1 => "Data_Control".AUTO."Auto.Mode1".STEP_E)
      Move(in := 0, out1 => "Data_Control".SlotIDTO)
      Move(in := 0, out1 => "Data_Control".AUTO."Auto.Mode2_Mode1".Step_ParkingCar)
   END_RUNG
   RUNG wire#w1
      { S7_Templates := "SrcType := Int" } EQ_Contact(in1 := "Data_Control".SlotIDTO, in2 := 202)
      S_Coil( "Data_Control".POSITION."202_C" )
      Move(in := 0, out1 => "Data_Control".AUTO."Auto.Mode1".STEP_E)
      Move(in := 0, out1 => "Data_Control".SlotIDTO)
      Move(in := 0, out1 => "Data_Control".AUTO."Auto.Mode2_Mode1".Step_ParkingCar)
   END_RUNG
   // the same network as SCL:
   #_w1 := "Data_Control".AUTO."Auto.Mode2_Mode1".Step_ParkingCar = 10;
   IF #_w1 AND ("Data_Control".SlotIDTO = 201) THEN
       "Data_Control".POSITION."201_C" := TRUE;
       "Data_Control".AUTO."Auto.Mode1".STEP_E := 0;
   END_IF;
   #_w2 := #_w1 AND ("Data_Control".SlotIDTO = 201);
   IF #_w2 THEN
       "Data_Control".SlotIDTO := 0;
       "Data_Control".AUTO."Auto.Mode2_Mode1".Step_ParkingCar := 0;
   END_IF;
   IF #_w1 AND ("Data_Control".SlotIDTO = 202) THEN
       "Data_Control".POSITION."202_C" := TRUE;
       "Data_Control".AUTO."Auto.Mode1".STEP_E := 0;
   END_IF;
   #_w3 := #_w1 AND ("Data_Control".SlotIDTO = 202);
   IF #_w3 THEN
       "Data_Control".SlotIDTO := 0;
       "Data_Control".AUTO."Auto.Mode2_Mode1".Step_ParkingCar := 0;
   END_IF;
END_REGION
END_FUNCTION_BLOCK

FUNCTION_BLOCK "ControlAtElevator"   // FB11, LAD
{ S7_Optimized_Access := 'FALSE' }
VERSION : 0.1
BEGIN

REGION Network 1
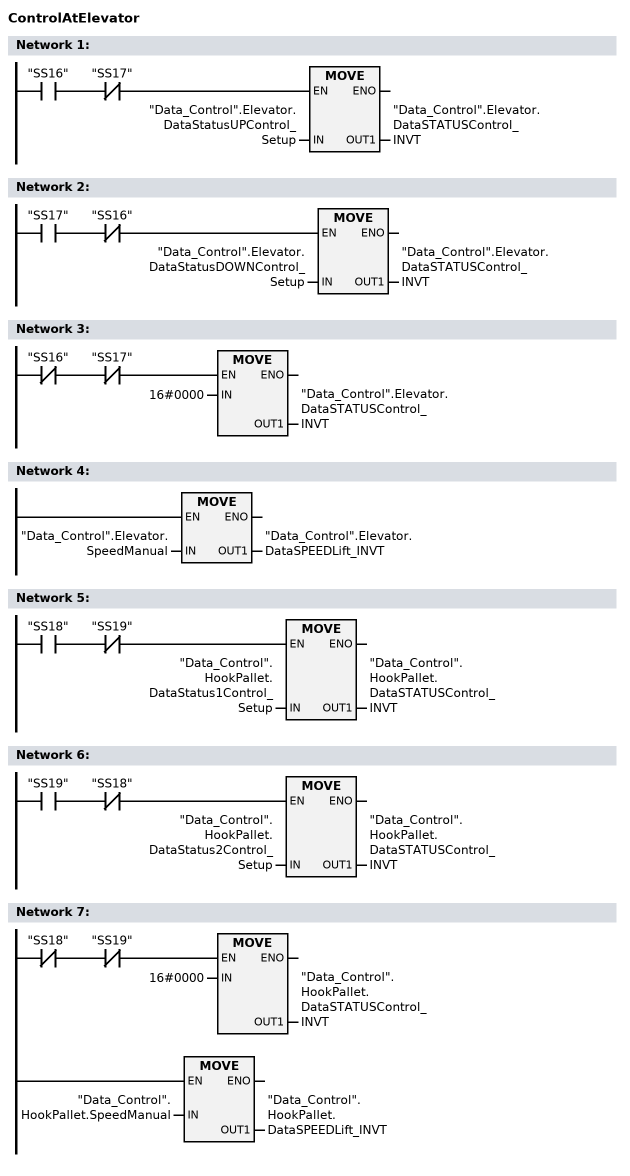
   RUNG wire#powerrail
      Contact( "SS16" )
      I_Contact( "SS17" )
      Move(in := "Data_Control".Elevator.DataStatusUPControl_Setup, out1 => "Data_Control".Elevator.DataSTATUSControl_INVT)
   END_RUNG
   // the same network as SCL:
   IF "SS16" AND NOT "SS17" THEN
       "Data_Control".Elevator.DataSTATUSControl_INVT := "Data_Control".Elevator.DataStatusUPControl_Setup;
   END_IF;
END_REGION

REGION Network 2
   RUNG wire#powerrail
      Contact( "SS17" )
      I_Contact( "SS16" )
      Move(in := "Data_Control".Elevator.DataStatusDOWNControl_Setup, out1 => "Data_Control".Elevator.DataSTATUSControl_INVT)
   END_RUNG
   // the same network as SCL:
   IF "SS17" AND NOT "SS16" THEN
       "Data_Control".Elevator.DataSTATUSControl_INVT := "Data_Control".Elevator.DataStatusDOWNControl_Setup;
   END_IF;
END_REGION

REGION Network 3
   RUNG wire#powerrail
      I_Contact( "SS16" )
      I_Contact( "SS17" )
      Move(in := 16#0000, out1 => "Data_Control".Elevator.DataSTATUSControl_INVT)
   END_RUNG
   // the same network as SCL:
   IF NOT "SS16" AND NOT "SS17" THEN "Data_Control".Elevator.DataSTATUSControl_INVT := 16#0000; END_IF;
END_REGION

REGION Network 4
   RUNG wire#powerrail
      Move(in := "Data_Control".Elevator.SpeedManual, out1 => "Data_Control".Elevator.DataSPEEDLift_INVT)
   END_RUNG
   // the same network as SCL:
   "Data_Control".Elevator.DataSPEEDLift_INVT := "Data_Control".Elevator.SpeedManual;
END_REGION

REGION Network 5
   RUNG wire#powerrail
      Contact( "SS18" )
      I_Contact( "SS19" )
      Move(in := "Data_Control".HookPallet.DataStatus1Control_Setup, out1 => "Data_Control".HookPallet.DataSTATUSControl_INVT)
   END_RUNG
   // the same network as SCL:
   IF "SS18" AND NOT "SS19" THEN
       "Data_Control".HookPallet.DataSTATUSControl_INVT := "Data_Control".HookPallet.DataStatus1Control_Setup;
   END_IF;
END_REGION

REGION Network 6
   RUNG wire#powerrail
      Contact( "SS19" )
      I_Contact( "SS18" )
      Move(in := "Data_Control".HookPallet.DataStatus2Control_Setup, out1 => "Data_Control".HookPallet.DataSTATUSControl_INVT)
   END_RUNG
   // the same network as SCL:
   IF "SS19" AND NOT "SS18" THEN
       "Data_Control".HookPallet.DataSTATUSControl_INVT := "Data_Control".HookPallet.DataStatus2Control_Setup;
   END_IF;
END_REGION

REGION Network 7
   RUNG wire#powerrail
      I_Contact( "SS18" )
      I_Contact( "SS19" )
      Move(in := 16#0000, out1 => "Data_Control".HookPallet.DataSTATUSControl_INVT)
   END_RUNG
   RUNG wire#powerrail
      Move(in := "Data_Control".HookPallet.SpeedManual, out1 => "Data_Control".HookPallet.DataSPEEDLift_INVT)
   END_RUNG
   // the same network as SCL:
   IF NOT "SS18" AND NOT "SS19" THEN "Data_Control".HookPallet.DataSTATUSControl_INVT := 16#0000; END_IF;
   "Data_Control".HookPallet.DataSPEEDLift_INVT := "Data_Control".HookPallet.SpeedManual;
END_REGION
END_FUNCTION_BLOCK

FUNCTION_BLOCK "ADMIN_HMI"   // FB12, LAD
{ S7_Optimized_Access := 'FALSE' }
VERSION : 0.1
   VAR_TEMP   // added for the SCL form of the ladder/FBD networks
      _w1 : Bool;
      _w2 : Bool;
   END_VAR
BEGIN

REGION Network 1
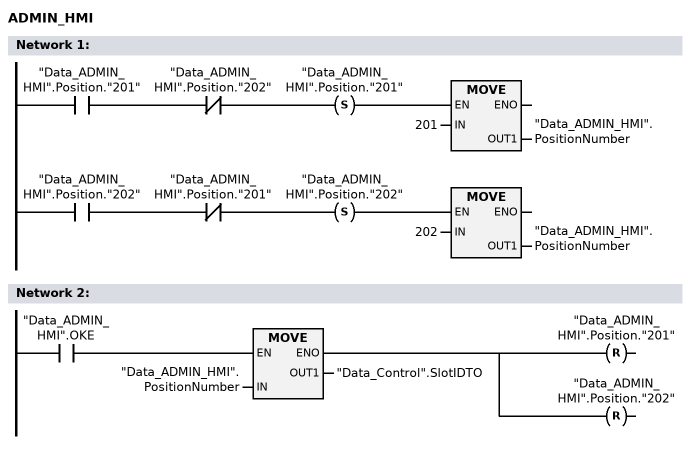
   RUNG wire#powerrail
      Contact( "Data_ADMIN_HMI".Position."201" )
      I_Contact( "Data_ADMIN_HMI".Position."202" )
      S_Coil( "Data_ADMIN_HMI".Position."201" )
      Move(in := 201, out1 => "Data_ADMIN_HMI".PositionNumber)
   END_RUNG
   RUNG wire#powerrail
      Contact( "Data_ADMIN_HMI".Position."202" )
      I_Contact( "Data_ADMIN_HMI".Position."201" )
      S_Coil( "Data_ADMIN_HMI".Position."202" )
      Move(in := 202, out1 => "Data_ADMIN_HMI".PositionNumber)
   END_RUNG
   // the same network as SCL:
   #_w1 := "Data_ADMIN_HMI".Position."201" AND NOT "Data_ADMIN_HMI".Position."202";
   IF #_w1 THEN
       "Data_ADMIN_HMI".Position."201" := TRUE;
       "Data_ADMIN_HMI".PositionNumber := 201;
   END_IF;
   #_w2 := "Data_ADMIN_HMI".Position."202" AND NOT "Data_ADMIN_HMI".Position."201";
   IF #_w2 THEN
       "Data_ADMIN_HMI".Position."202" := TRUE;
       "Data_ADMIN_HMI".PositionNumber := 202;
   END_IF;
END_REGION

REGION Network 2
   RUNG wire#powerrail
      Contact( "Data_ADMIN_HMI".OKE )
      Move(in := "Data_ADMIN_HMI".PositionNumber, out1 => "Data_Control".SlotIDTO)
      wire#w1
      R_Coil( "Data_ADMIN_HMI".Position."201" )
   END_RUNG
   RUNG wire#w1
      R_Coil( "Data_ADMIN_HMI".Position."202" )
   END_RUNG
   // the same network as SCL:
   IF "Data_ADMIN_HMI".OKE THEN
       "Data_Control".SlotIDTO := "Data_ADMIN_HMI".PositionNumber;
       "Data_ADMIN_HMI".Position."201" := FALSE;
       "Data_ADMIN_HMI".Position."202" := FALSE;
   END_IF;
END_REGION
END_FUNCTION_BLOCK

FUNCTION_BLOCK "POSITION"   // FB13, LAD
{ S7_Optimized_Access := 'TRUE' }
VERSION : 0.1
BEGIN

REGION Network 1
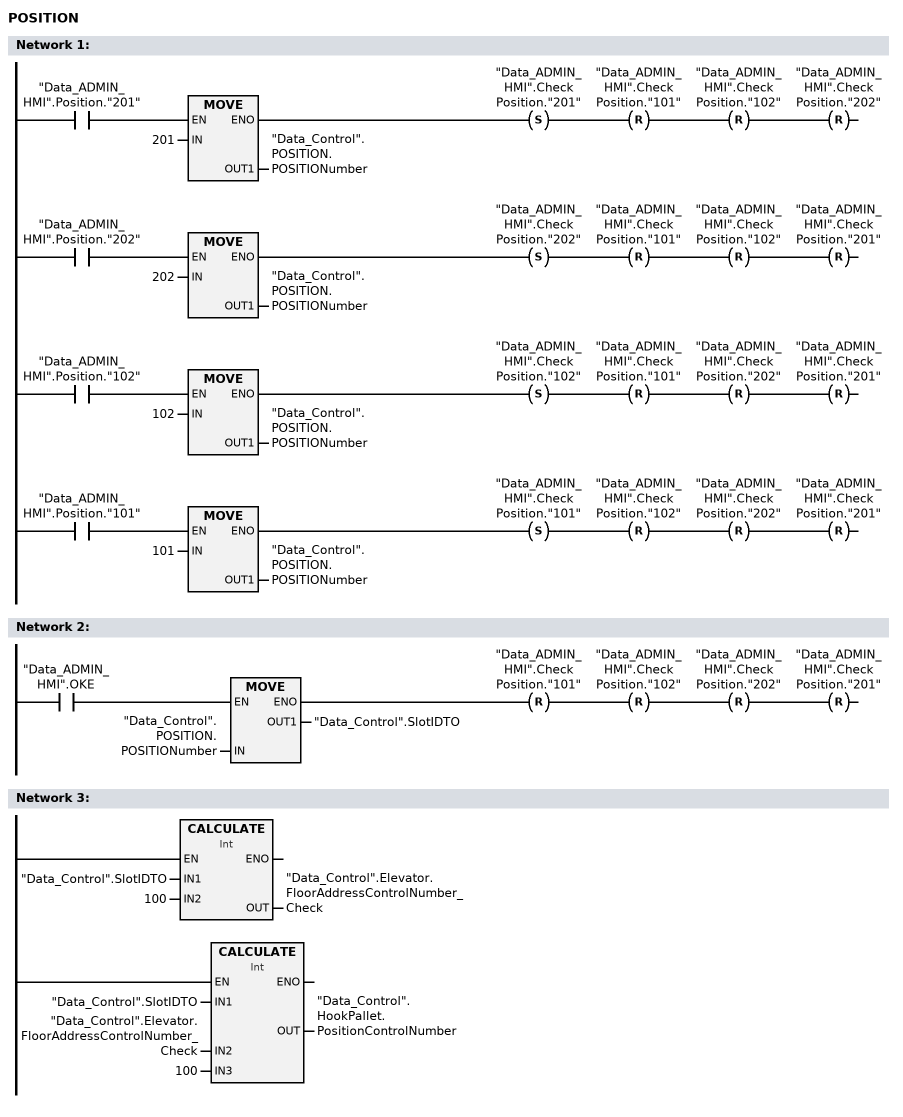
   RUNG wire#powerrail
      Contact( "Data_ADMIN_HMI".Position."201" )
      Move(in := 201, out1 => "Data_Control".POSITION.POSITIONumber)
      S_Coil( "Data_ADMIN_HMI".CheckPosition."201" )
      R_Coil( "Data_ADMIN_HMI".CheckPosition."101" )
      R_Coil( "Data_ADMIN_HMI".CheckPosition."102" )
      R_Coil( "Data_ADMIN_HMI".CheckPosition."202" )
   END_RUNG
   RUNG wire#powerrail
      Contact( "Data_ADMIN_HMI".Position."202" )
      Move(in := 202, out1 => "Data_Control".POSITION.POSITIONumber)
      S_Coil( "Data_ADMIN_HMI".CheckPosition."202" )
      R_Coil( "Data_ADMIN_HMI".CheckPosition."101" )
      R_Coil( "Data_ADMIN_HMI".CheckPosition."102" )
      R_Coil( "Data_ADMIN_HMI".CheckPosition."201" )
   END_RUNG
   RUNG wire#powerrail
      Contact( "Data_ADMIN_HMI".Position."102" )
      Move(in := 102, out1 => "Data_Control".POSITION.POSITIONumber)
      S_Coil( "Data_ADMIN_HMI".CheckPosition."102" )
      R_Coil( "Data_ADMIN_HMI".CheckPosition."101" )
      R_Coil( "Data_ADMIN_HMI".CheckPosition."202" )
      R_Coil( "Data_ADMIN_HMI".CheckPosition."201" )
   END_RUNG
   RUNG wire#powerrail
      Contact( "Data_ADMIN_HMI".Position."101" )
      Move(in := 101, out1 => "Data_Control".POSITION.POSITIONumber)
      S_Coil( "Data_ADMIN_HMI".CheckPosition."101" )
      R_Coil( "Data_ADMIN_HMI".CheckPosition."102" )
      R_Coil( "Data_ADMIN_HMI".CheckPosition."202" )
      R_Coil( "Data_ADMIN_HMI".CheckPosition."201" )
   END_RUNG
   // the same network as SCL:
   IF "Data_ADMIN_HMI".Position."201" THEN
       "Data_Control".POSITION.POSITIONumber := 201;
       "Data_ADMIN_HMI".CheckPosition."201" := TRUE;
       "Data_ADMIN_HMI".CheckPosition."101" := FALSE;
       "Data_ADMIN_HMI".CheckPosition."102" := FALSE;
       "Data_ADMIN_HMI".CheckPosition."202" := FALSE;
   END_IF;
   IF "Data_ADMIN_HMI".Position."202" THEN
       "Data_Control".POSITION.POSITIONumber := 202;
       "Data_ADMIN_HMI".CheckPosition."202" := TRUE;
       "Data_ADMIN_HMI".CheckPosition."101" := FALSE;
       "Data_ADMIN_HMI".CheckPosition."102" := FALSE;
       "Data_ADMIN_HMI".CheckPosition."201" := FALSE;
   END_IF;
   IF "Data_ADMIN_HMI".Position."102" THEN
       "Data_Control".POSITION.POSITIONumber := 102;
       "Data_ADMIN_HMI".CheckPosition."102" := TRUE;
       "Data_ADMIN_HMI".CheckPosition."101" := FALSE;
       "Data_ADMIN_HMI".CheckPosition."202" := FALSE;
       "Data_ADMIN_HMI".CheckPosition."201" := FALSE;
   END_IF;
   IF "Data_ADMIN_HMI".Position."101" THEN
       "Data_Control".POSITION.POSITIONumber := 101;
       "Data_ADMIN_HMI".CheckPosition."101" := TRUE;
       "Data_ADMIN_HMI".CheckPosition."102" := FALSE;
       "Data_ADMIN_HMI".CheckPosition."202" := FALSE;
       "Data_ADMIN_HMI".CheckPosition."201" := FALSE;
   END_IF;
END_REGION

REGION Network 2
   RUNG wire#powerrail
      Contact( "Data_ADMIN_HMI".OKE )
      Move(in := "Data_Control".POSITION.POSITIONumber, out1 => "Data_Control".SlotIDTO)
      R_Coil( "Data_ADMIN_HMI".CheckPosition."101" )
      R_Coil( "Data_ADMIN_HMI".CheckPosition."102" )
      R_Coil( "Data_ADMIN_HMI".CheckPosition."202" )
      R_Coil( "Data_ADMIN_HMI".CheckPosition."201" )
   END_RUNG
   // the same network as SCL:
   IF "Data_ADMIN_HMI".OKE THEN
       "Data_Control".SlotIDTO := "Data_Control".POSITION.POSITIONumber;
       "Data_ADMIN_HMI".CheckPosition."101" := FALSE;
       "Data_ADMIN_HMI".CheckPosition."102" := FALSE;
       "Data_ADMIN_HMI".CheckPosition."202" := FALSE;
       "Data_ADMIN_HMI".CheckPosition."201" := FALSE;
   END_IF;
END_REGION

REGION Network 3
   RUNG wire#powerrail
      { S7_Templates := "SrcType := Int"; S7_Expression := "IN1/IN2" } Calculate(in1 := "Data_Control".SlotIDTO, in2 := 100, out => "Data_Control".Elevator.FloorAddressControlNumber_Check)
   END_RUNG
   RUNG wire#powerrail
      { S7_Templates := "SrcType := Int"; S7_Expression := "IN1-(IN2*IN3)" } Calculate(in1 := "Data_Control".SlotIDTO, in2 := "Data_Control".Elevator.FloorAddressControlNumber_Check, in3 := 100, out => "Data_Control".HookPallet.PositionControlNumber)
   END_RUNG
   // the same network as SCL:
   "Data_Control".Elevator.FloorAddressControlNumber_Check := "Data_Control".SlotIDTO/100;
   "Data_Control".HookPallet.PositionControlNumber := "Data_Control".SlotIDTO-("Data_Control".Elevator.FloorAddressControlNumber_Check*100);
END_REGION
END_FUNCTION_BLOCK

ORGANIZATION_BLOCK "Main"   // OB1, LAD, ProgramCycle
TITLE = "Main Program Sweep (Cycle)"
{ S7_Optimized_Access := 'TRUE' }
VERSION : 0.1
   VAR_INPUT
      Initial_Call : Bool;   // Initial call of this OB
      Remanence : Bool;   // =True, if remanent data are available
   END_VAR
BEGIN

REGION Network 1
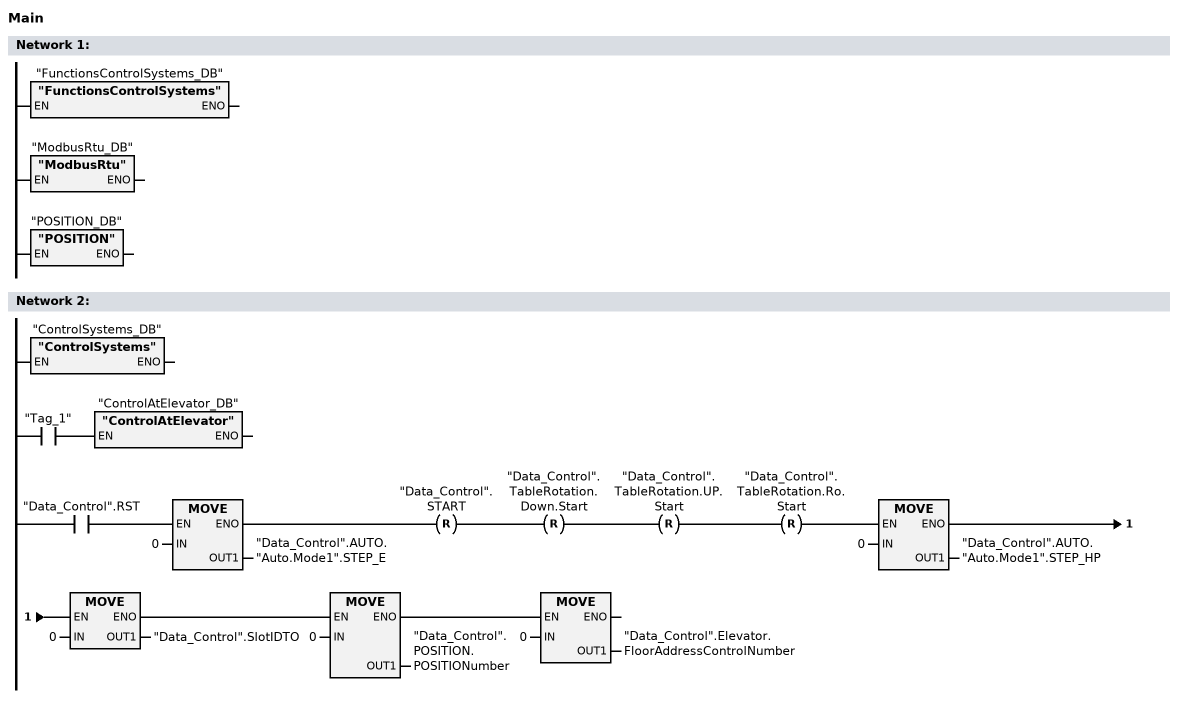
   RUNG wire#powerrail
      "FunctionsControlSystems_DB"()
   END_RUNG
   RUNG wire#powerrail
      "ModbusRtu_DB"()
   END_RUNG
   RUNG wire#powerrail
      "POSITION_DB"()
   END_RUNG
   // the same network as SCL:
   "FunctionsControlSystems_DB"();   // "FunctionsControlSystems"
   "ModbusRtu_DB"();   // "ModbusRtu"
   "POSITION_DB"();   // "POSITION"
END_REGION

REGION Network 2
   RUNG wire#powerrail
      "ControlSystems_DB"()
   END_RUNG
   RUNG wire#powerrail
      Contact( "Tag_1" )
      "ControlAtElevator_DB"()
   END_RUNG
   RUNG wire#powerrail
      Contact( "Data_Control".RST )
      Move(in := 0, out1 => "Data_Control".AUTO."Auto.Mode1".STEP_E)
      R_Coil( "Data_Control".START )
      R_Coil( "Data_Control".TableRotation.Down.Start )
      R_Coil( "Data_Control".TableRotation.UP.Start )
      R_Coil( "Data_Control".TableRotation.Ro.Start )
      Move(in := 0, out1 => "Data_Control".AUTO."Auto.Mode1".STEP_HP)
      Move(in := 0, out1 => "Data_Control".SlotIDTO)
      Move(in := 0, out1 => "Data_Control".POSITION.POSITIONumber)
      Move(in := 0, out1 => "Data_Control".Elevator.FloorAddressControlNumber)
   END_RUNG
   // the same network as SCL:
   "ControlSystems_DB"();   // "ControlSystems"
   IF "Tag_1" THEN
       "ControlAtElevator_DB"();   // "ControlAtElevator"
   END_IF;
   IF "Data_Control".RST THEN
       "Data_Control".AUTO."Auto.Mode1".STEP_E := 0;
       "Data_Control".START := FALSE;
       "Data_Control".TableRotation.Down.Start := FALSE;
       "Data_Control".TableRotation.UP.Start := FALSE;
       "Data_Control".TableRotation.Ro.Start := FALSE;
       "Data_Control".AUTO."Auto.Mode1".STEP_HP := 0;
       "Data_Control".SlotIDTO := 0;
       "Data_Control".POSITION.POSITIONumber := 0;
       "Data_Control".Elevator.FloorAddressControlNumber := 0;
   END_IF;
END_REGION
END_ORGANIZATION_BLOCK

// folder: Control/FunctionsControlSystem

FUNCTION_BLOCK "ElevatorMcFullFunction"   // FB24, LAD
{ S7_Optimized_Access := 'FALSE' }
VERSION : 0.1
   VAR_INPUT
      Manual_Auto : Bool;
      START : Bool;
      STOP : Bool;
      UP : Bool;
      ERROR : Bool;
      DOWN : Bool;
      RST : Bool;
      Sensor_Count_Floor : Bool;
      Sensor_Count_Floor_Check : Bool;
      Sensor_Stop : Bool;
      Speed_Manual : Int;
      Speed_Startup : Int;
      "time 1" : Time;
      Speed1_Auto : Int;
      "time 2" : Time;
      Speed2_Auto : Int;
      "time 3" : Time;
      Speed_Stop_Auto : Int;
   END_VAR
   VAR_OUTPUT
      Done_LIFT : Bool;
      Running : Bool;   // Lift Running
      FLOOR_ADDRESS_REAL : Int := 1;   // address Elevator standing
      FLOOR_ADDRESS_REAL_Check : Int := 1;
      "FLOOR_ADDRESS_REAL SUB  FLOOR_ADDRESS_CONTROLL_NUMBER" : Int;
      Data_Speed_Running : Int;
      Data_Status_INVT_Modbus : Word;   // Data use to Modbus RTU
      FromID : Int;
   END_VAR
   VAR_IN_OUT
      Step_LIFT : Int;   // steps used to control
      STATUS_Run_Up : Word;   // Set_Up Run R/F
      STATUS_Run_DOWN : Word;   // Set_Up Run R/F
      FLOOR_ADDRESS_CONTROLL_NUMBER : Int;
   END_VAR
   VAR_TEMP   // added for the SCL form of the ladder/FBD networks
      _w1 : Bool;
      _w2 : Bool;
   END_VAR
BEGIN

REGION Network 1
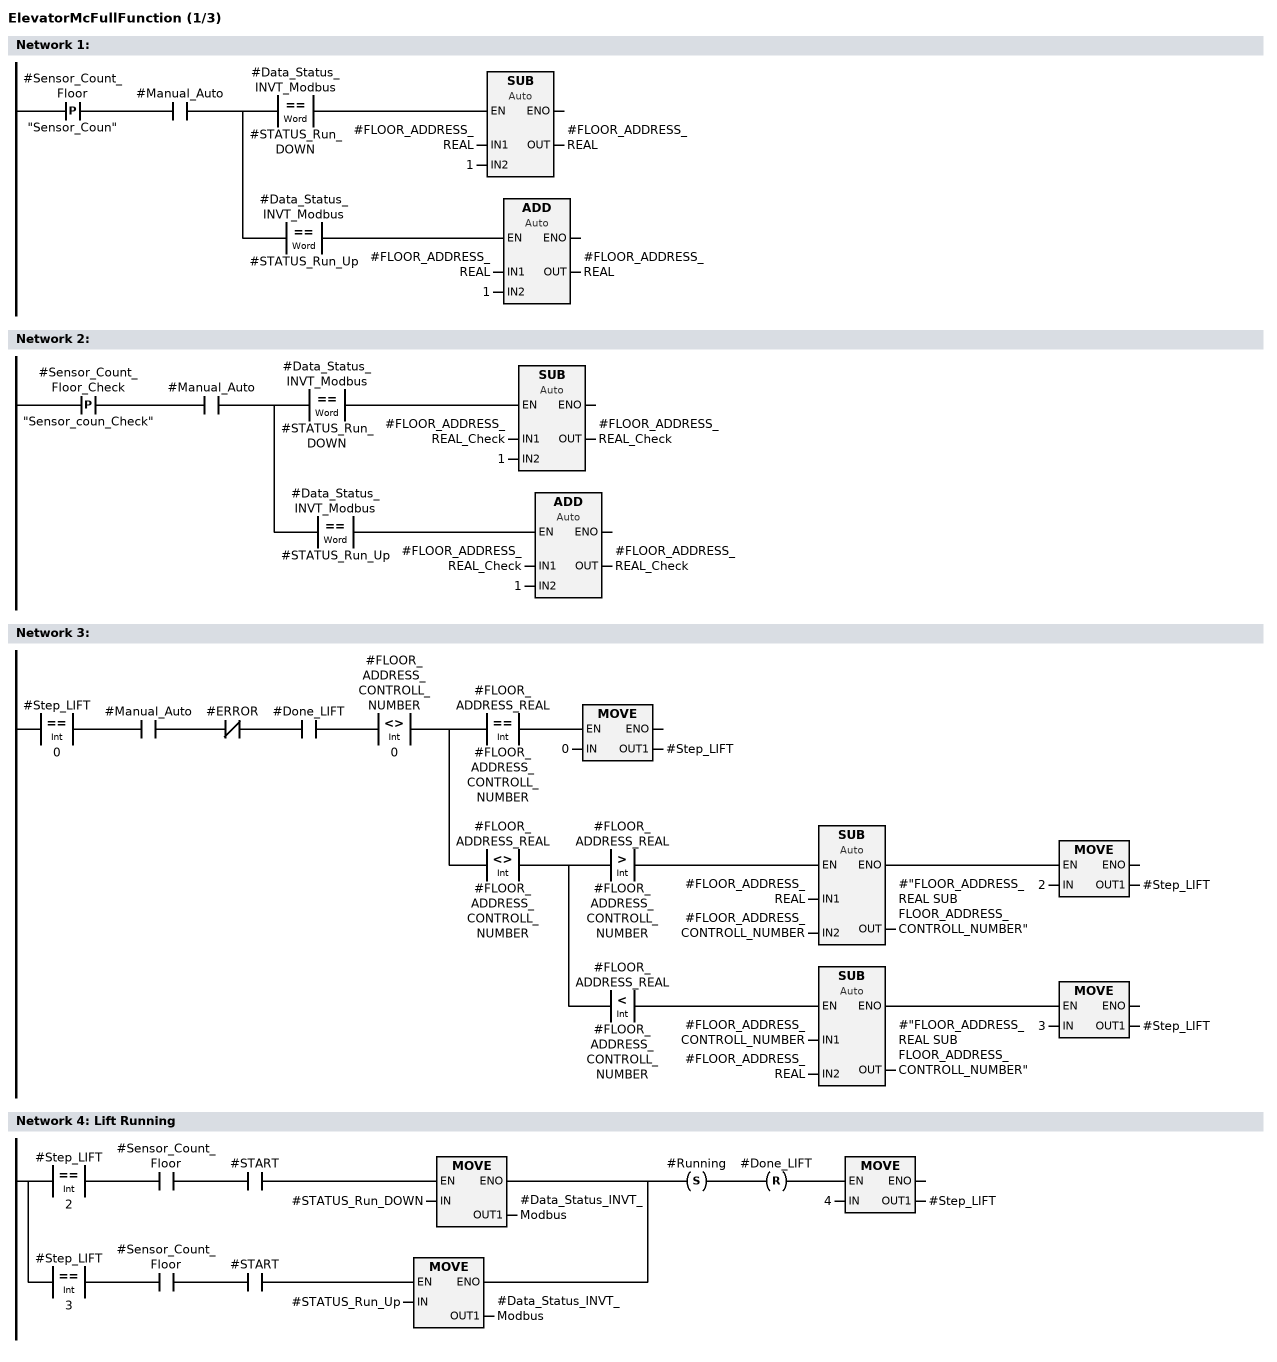
   RUNG wire#powerrail
      P_Contact(operand := #Sensor_Count_Floor, bit := "Sensor_Coun")
      Contact( #Manual_Auto )
      wire#w1
      { S7_Templates := "SrcType := Word" } EQ_Contact(in1 := #Data_Status_INVT_Modbus, in2 := #STATUS_Run_DOWN)
      Sub(in1 := #FLOOR_ADDRESS_REAL, in2 := 1, out => #FLOOR_ADDRESS_REAL)
   END_RUNG
   RUNG wire#w1
      { S7_Templates := "SrcType := Word" } EQ_Contact(in1 := #Data_Status_INVT_Modbus, in2 := #STATUS_Run_Up)
      Add(in1 := #FLOOR_ADDRESS_REAL, in2 := 1, out => #FLOOR_ADDRESS_REAL)
   END_RUNG
   // the same network as SCL:
   #_w1 := #Sensor_Count_Floor AND NOT "Sensor_Coun";   // rising edge of #Sensor_Count_Floor
   "Sensor_Coun" := #Sensor_Count_Floor;
   #_w2 := #_w1 AND #Manual_Auto;
   IF #_w2 AND (#Data_Status_INVT_Modbus = #STATUS_Run_DOWN) THEN
       #FLOOR_ADDRESS_REAL := #FLOOR_ADDRESS_REAL - 1;
   END_IF;
   IF #_w2 AND (#Data_Status_INVT_Modbus = #STATUS_Run_Up) THEN
       #FLOOR_ADDRESS_REAL := #FLOOR_ADDRESS_REAL + 1;
   END_IF;
END_REGION

REGION Network 2
   RUNG wire#powerrail
      P_Contact(operand := #Sensor_Count_Floor_Check, bit := "Sensor_coun_Check")
      Contact( #Manual_Auto )
      wire#w1
      { S7_Templates := "SrcType := Word" } EQ_Contact(in1 := #Data_Status_INVT_Modbus, in2 := #STATUS_Run_DOWN)
      Sub(in1 := #FLOOR_ADDRESS_REAL_Check, in2 := 1, out => #FLOOR_ADDRESS_REAL_Check)
   END_RUNG
   RUNG wire#w1
      { S7_Templates := "SrcType := Word" } EQ_Contact(in1 := #Data_Status_INVT_Modbus, in2 := #STATUS_Run_Up)
      Add(in1 := #FLOOR_ADDRESS_REAL_Check, in2 := 1, out => #FLOOR_ADDRESS_REAL_Check)
   END_RUNG
   // the same network as SCL:
   #_w1 := #Sensor_Count_Floor_Check AND NOT "Sensor_coun_Check";   // rising edge of #Sensor_Count_Floor_Check
   "Sensor_coun_Check" := #Sensor_Count_Floor_Check;
   #_w2 := #_w1 AND #Manual_Auto;
   IF #_w2 AND (#Data_Status_INVT_Modbus = #STATUS_Run_DOWN) THEN
       #FLOOR_ADDRESS_REAL_Check := #FLOOR_ADDRESS_REAL_Check - 1;
   END_IF;
   IF #_w2 AND (#Data_Status_INVT_Modbus = #STATUS_Run_Up) THEN
       #FLOOR_ADDRESS_REAL_Check := #FLOOR_ADDRESS_REAL_Check + 1;
   END_IF;
END_REGION

REGION Network 3
   RUNG wire#powerrail
      { S7_Templates := "SrcType := Int" } EQ_Contact(in1 := #Step_LIFT, in2 := 0)
      Contact( #Manual_Auto )
      I_Contact( #ERROR )
      Contact( #Done_LIFT )
      { S7_Templates := "SrcType := Int" } NE_Contact(in1 := #FLOOR_ADDRESS_CONTROLL_NUMBER, in2 := 0)
      wire#w1
      { S7_Templates := "SrcType := Int" } EQ_Contact(in1 := #FLOOR_ADDRESS_REAL, in2 := #FLOOR_ADDRESS_CONTROLL_NUMBER)
      Move(in := 0, out1 => #Step_LIFT)
   END_RUNG
   RUNG wire#w1
      { S7_Templates := "SrcType := Int" } NE_Contact(in1 := #FLOOR_ADDRESS_REAL, in2 := #FLOOR_ADDRESS_CONTROLL_NUMBER)
      wire#w2
      { S7_Templates := "SrcType := Int" } GT_Contact(in1 := #FLOOR_ADDRESS_REAL, in2 := #FLOOR_ADDRESS_CONTROLL_NUMBER)
      Sub(in1 := #FLOOR_ADDRESS_REAL, in2 := #FLOOR_ADDRESS_CONTROLL_NUMBER, out => #"FLOOR_ADDRESS_REAL SUB  FLOOR_ADDRESS_CONTROLL_NUMBER")
      Move(in := 2, out1 => #Step_LIFT)
   END_RUNG
   RUNG wire#w2
      { S7_Templates := "SrcType := Int" } LT_Contact(in1 := #FLOOR_ADDRESS_REAL, in2 := #FLOOR_ADDRESS_CONTROLL_NUMBER)
      Sub(in1 := #FLOOR_ADDRESS_CONTROLL_NUMBER, in2 := #FLOOR_ADDRESS_REAL, out => #"FLOOR_ADDRESS_REAL SUB  FLOOR_ADDRESS_CONTROLL_NUMBER")
      Move(in := 3, out1 => #Step_LIFT)
   END_RUNG
   // the same network as SCL:
   #_w1 := (#Step_LIFT = 0) AND #Manual_Auto AND NOT #ERROR AND #Done_LIFT AND (#FLOOR_ADDRESS_CONTROLL_NUMBER <> 0);
   IF #_w1 AND (#FLOOR_ADDRESS_REAL = #FLOOR_ADDRESS_CONTROLL_NUMBER) THEN #Step_LIFT := 0; END_IF;
   #_w2 := #_w1 AND (#FLOOR_ADDRESS_REAL <> #FLOOR_ADDRESS_CONTROLL_NUMBER);
   IF #_w2 AND (#FLOOR_ADDRESS_REAL > #FLOOR_ADDRESS_CONTROLL_NUMBER) THEN
       #"FLOOR_ADDRESS_REAL SUB  FLOOR_ADDRESS_CONTROLL_NUMBER" := #FLOOR_ADDRESS_REAL - #FLOOR_ADDRESS_CONTROLL_NUMBER;
       #Step_LIFT := 2;
   END_IF;
   IF #_w2 AND (#FLOOR_ADDRESS_REAL < #FLOOR_ADDRESS_CONTROLL_NUMBER) THEN
       #"FLOOR_ADDRESS_REAL SUB  FLOOR_ADDRESS_CONTROLL_NUMBER" := #FLOOR_ADDRESS_CONTROLL_NUMBER - #FLOOR_ADDRESS_REAL;
       #Step_LIFT := 3;
   END_IF;
END_REGION

REGION Network 4: Lift Running
   RUNG wire#powerrail
      { S7_Templates := "SrcType := Int" } EQ_Contact(in1 := #Step_LIFT, in2 := 2)
      Contact( #Sensor_Count_Floor )
      Contact( #START )
      Move(in := #STATUS_Run_DOWN, out1 => #Data_Status_INVT_Modbus)
      wire#w1
      S_Coil( #Running )
      R_Coil( #Done_LIFT )
      Move(in := 4, out1 => #Step_LIFT)
   END_RUNG
   RUNG wire#powerrail
      { S7_Templates := "SrcType := Int" } EQ_Contact(in1 := #Step_LIFT, in2 := 3)
      Contact( #Sensor_Count_Floor )
      Contact( #START )
      Move(in := #STATUS_Run_Up, out1 => #Data_Status_INVT_Modbus)
   END_RUNG wire#w1
   // the same network as SCL:
   #_w1 := (#Step_LIFT = 2) AND #Sensor_Count_Floor AND #START;
   IF #_w1 THEN #Data_Status_INVT_Modbus := #STATUS_Run_DOWN; END_IF;
   #_w2 := (#Step_LIFT = 3) AND #Sensor_Count_Floor AND #START;
   IF #_w2 THEN #Data_Status_INVT_Modbus := #STATUS_Run_Up; END_IF;
   IF #_w1 OR #_w2 THEN
       #Running := TRUE;
       #Done_LIFT := FALSE;
       #Step_LIFT := 4;
   END_IF;
END_REGION

REGION Network 5
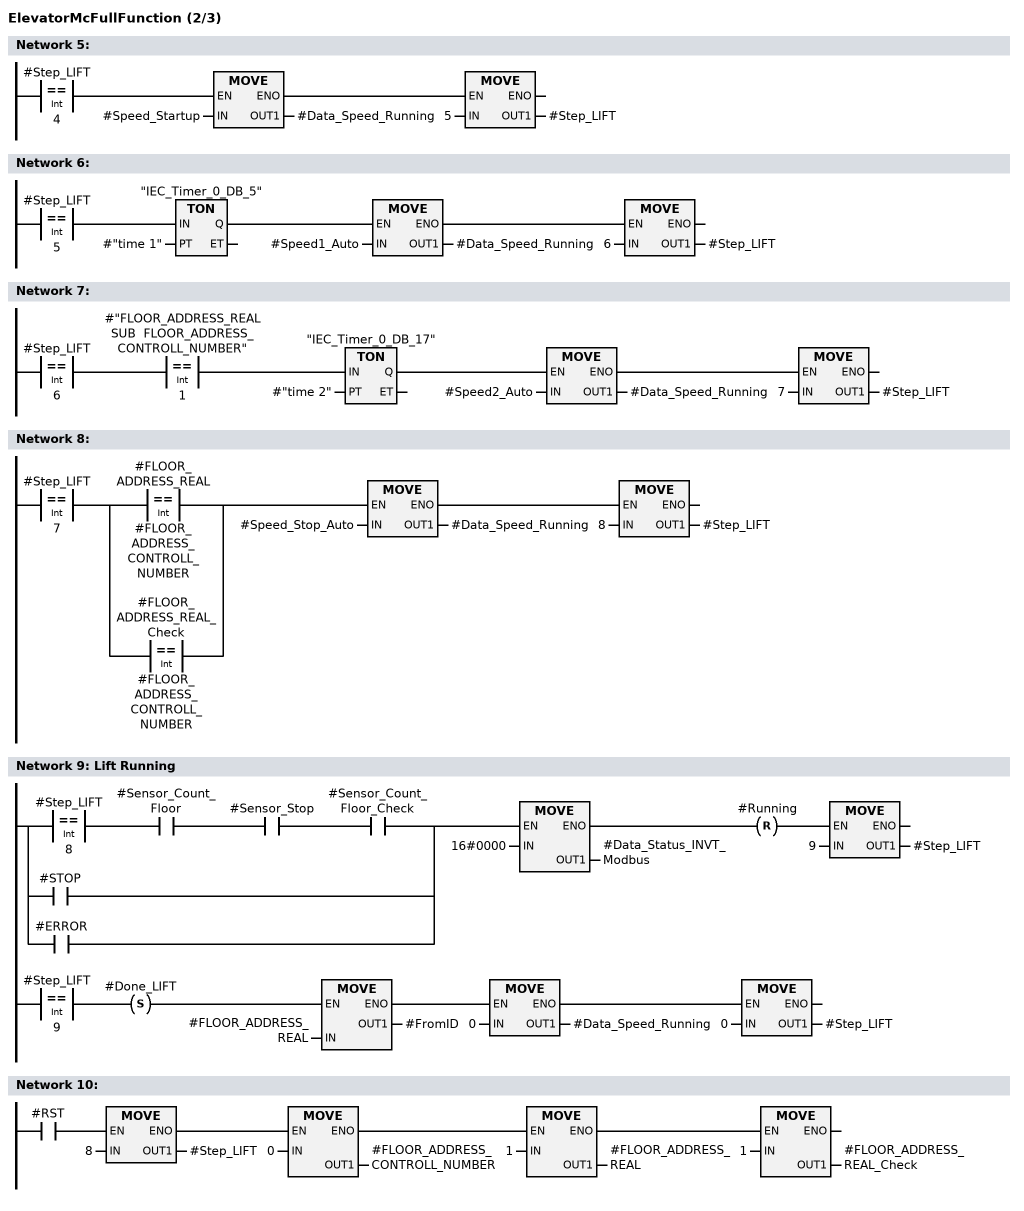
   RUNG wire#powerrail
      { S7_Templates := "SrcType := Int" } EQ_Contact(in1 := #Step_LIFT, in2 := 4)
      Move(in := #Speed_Startup, out1 => #Data_Speed_Running)
      Move(in := 5, out1 => #Step_LIFT)
   END_RUNG
   // the same network as SCL:
   IF #Step_LIFT = 4 THEN
       #Data_Speed_Running := #Speed_Startup;
       #Step_LIFT := 5;
   END_IF;
END_REGION

REGION Network 6
   "IEC_Timer_0_DB_5".TON(IN := #Step_LIFT = 5, PT := #"time 1");
   IF "IEC_Timer_0_DB_5".Q THEN
       #Data_Speed_Running := #Speed1_Auto;
       #Step_LIFT := 6;
   END_IF;
END_REGION

REGION Network 7
   "IEC_Timer_0_DB_17".TON(IN := (#Step_LIFT = 6) AND (#"FLOOR_ADDRESS_REAL SUB  FLOOR_ADDRESS_CONTROLL_NUMBER" = 1),
                           PT := #"time 2");
   IF "IEC_Timer_0_DB_17".Q THEN
       #Data_Speed_Running := #Speed2_Auto;
       #Step_LIFT := 7;
   END_IF;
END_REGION

REGION Network 8
   RUNG wire#powerrail
      { S7_Templates := "SrcType := Int" } EQ_Contact(in1 := #Step_LIFT, in2 := 7)
      wire#w1
      { S7_Templates := "SrcType := Int" } EQ_Contact(in1 := #FLOOR_ADDRESS_REAL, in2 := #FLOOR_ADDRESS_CONTROLL_NUMBER)
      wire#w2
      Move(in := #Speed_Stop_Auto, out1 => #Data_Speed_Running)
      Move(in := 8, out1 => #Step_LIFT)
   END_RUNG
   RUNG wire#w1
      { S7_Templates := "SrcType := Int" } EQ_Contact(in1 := #FLOOR_ADDRESS_REAL_Check, in2 := #FLOOR_ADDRESS_CONTROLL_NUMBER)
   END_RUNG wire#w2
   // the same network as SCL:
   IF (#Step_LIFT = 7) AND ((#FLOOR_ADDRESS_REAL = #FLOOR_ADDRESS_CONTROLL_NUMBER) OR (#FLOOR_ADDRESS_REAL_Check = #FLOOR_ADDRESS_CONTROLL_NUMBER)) THEN
       #Data_Speed_Running := #Speed_Stop_Auto;
       #Step_LIFT := 8;
   END_IF;
END_REGION

REGION Network 9: Lift Running
   RUNG wire#powerrail
      { S7_Templates := "SrcType := Int" } EQ_Contact(in1 := #Step_LIFT, in2 := 8)
      Contact( #Sensor_Count_Floor )
      Contact( #Sensor_Stop )
      Contact( #Sensor_Count_Floor_Check )
      wire#w1
      Move(in := 16#0000, out1 => #Data_Status_INVT_Modbus)
      R_Coil( #Running )
      Move(in := 9, out1 => #Step_LIFT)
   END_RUNG
   RUNG wire#powerrail
      Contact( #STOP )
   END_RUNG wire#w1
   RUNG wire#powerrail
      Contact( #ERROR )
   END_RUNG wire#w1
   RUNG wire#powerrail
      { S7_Templates := "SrcType := Int" } EQ_Contact(in1 := #Step_LIFT, in2 := 9)
      S_Coil( #Done_LIFT )
      Move(in := #FLOOR_ADDRESS_REAL, out1 => #FromID)
      Move(in := 0, out1 => #Data_Speed_Running)
      Move(in := 0, out1 => #Step_LIFT)
   END_RUNG
   // the same network as SCL:
   IF ((#Step_LIFT = 8) AND #Sensor_Count_Floor AND #Sensor_Stop AND #Sensor_Count_Floor_Check) OR #STOP OR #ERROR THEN
       #Data_Status_INVT_Modbus := 16#0000;
       #Running := FALSE;
       #Step_LIFT := 9;
   END_IF;
   IF #Step_LIFT = 9 THEN
       #Done_LIFT := TRUE;
       #FromID := #FLOOR_ADDRESS_REAL;
       #Data_Speed_Running := 0;
       #Step_LIFT := 0;
   END_IF;
END_REGION

REGION Network 10
   RUNG wire#powerrail
      Contact( #RST )
      Move(in := 8, out1 => #Step_LIFT)
      Move(in := 0, out1 => #FLOOR_ADDRESS_CONTROLL_NUMBER)
      Move(in := 1, out1 => #FLOOR_ADDRESS_REAL)
      Move(in := 1, out1 => #FLOOR_ADDRESS_REAL_Check)
   END_RUNG
   // the same network as SCL:
   IF #RST THEN
       #Step_LIFT := 8;
       #FLOOR_ADDRESS_CONTROLL_NUMBER := 0;
       #FLOOR_ADDRESS_REAL := 1;
       #FLOOR_ADDRESS_REAL_Check := 1;
   END_IF;
END_REGION

REGION Network 11: Control manual Lift Running
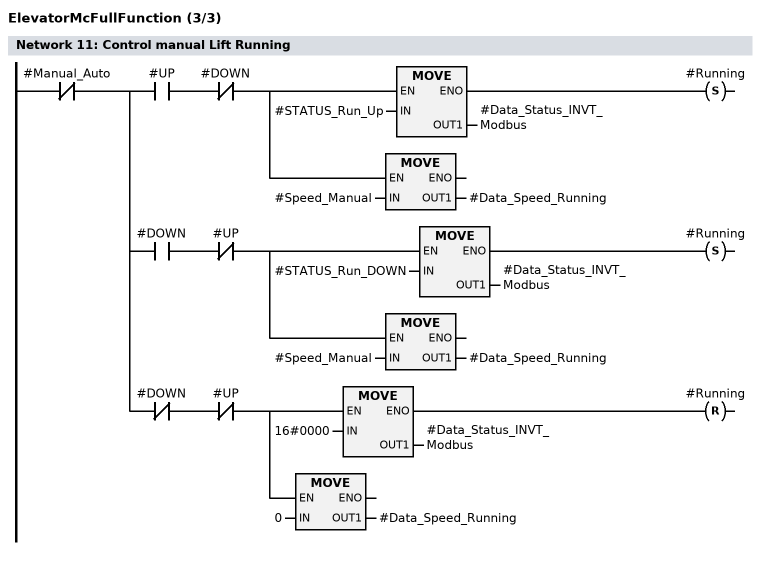
   RUNG wire#powerrail
      I_Contact( #Manual_Auto )
      wire#w1
      Contact( #UP )
      I_Contact( #DOWN )
      wire#w2
      Move(in := #STATUS_Run_Up, out1 => #Data_Status_INVT_Modbus)
      S_Coil( #Running )
   END_RUNG
   RUNG wire#w2
      Move(in := #Speed_Manual, out1 => #Data_Speed_Running)
   END_RUNG
   RUNG wire#w1
      Contact( #DOWN )
      I_Contact( #UP )
      wire#w3
      Move(in := #STATUS_Run_DOWN, out1 => #Data_Status_INVT_Modbus)
      S_Coil( #Running )
   END_RUNG
   RUNG wire#w3
      Move(in := #Speed_Manual, out1 => #Data_Speed_Running)
   END_RUNG
   RUNG wire#w1
      I_Contact( #DOWN )
      I_Contact( #UP )
      wire#w4
      Move(in := 16#0000, out1 => #Data_Status_INVT_Modbus)
      R_Coil( #Running )
   END_RUNG
   RUNG wire#w4
      Move(in := 0, out1 => #Data_Speed_Running)
   END_RUNG
   // the same network as SCL:
   IF NOT #Manual_Auto AND #UP AND NOT #DOWN THEN
       #Data_Status_INVT_Modbus := #STATUS_Run_Up;
       #Running := TRUE;
       #Data_Speed_Running := #Speed_Manual;
   END_IF;
   IF NOT #Manual_Auto AND #DOWN AND NOT #UP THEN
       #Data_Status_INVT_Modbus := #STATUS_Run_DOWN;
       #Running := TRUE;
       #Data_Speed_Running := #Speed_Manual;
   END_IF;
   IF NOT #Manual_Auto AND NOT #DOWN AND NOT #UP THEN
       #Data_Status_INVT_Modbus := 16#0000;
       #Running := FALSE;
       #Data_Speed_Running := 0;
   END_IF;
END_REGION
END_FUNCTION_BLOCK

FUNCTION_BLOCK "FunctionsControlSystems"   // FB26, LAD
{ S7_Optimized_Access := 'TRUE' }
VERSION : 0.1
   VAR_TEMP   // added for the SCL form of the ladder/FBD networks
      _w1 : Bool;
      _w2 : Bool;
   END_VAR
BEGIN

